// TwinCAT 3 PLC project PLC
// ProgramVersion: 3.1.4026.21
// libraries:
//   Core, * (Beckhoff Automation LLC)
//   CoreComponents, * (Beckhoff Automation LLC)
//   CoreMotionNc2, * (Beckhoff Automation LLC)
//   Tc2_ControllerToolbox, * (Beckhoff Automation GmbH)
//   Tc2_EtherCAT, * (Beckhoff Automation GmbH)
//   Tc2_MC2, * (Beckhoff Automation GmbH)
//   Tc2_Standard, * (Beckhoff Automation GmbH)
//   Tc2_System, * (Beckhoff Automation GmbH)
//   Tc2_TcpIp, * (Beckhoff Automation GmbH)
//   Tc3_JsonXml, * (Beckhoff Automation GmbH)
//   Tc3_PackML_V3, * (Beckhoff Automation GmbH)
// project tree:
//   AMR/ AMR_CONSTANT.TcGVL, AmrModule.TcPOU, AmrModule_HMI.TcPOU
//   AMR/DUT/ ST_AxisRecipe.TcDUT, ST_Recipe.TcDUT, ST_AmrModule_HMI.TcDUT
//   AMR/Interface/ I_AmrModule.TcIO
//   Components/Accelerometer %28EP3751%29/DUT/ ST_EP3751.TcDUT (not stored), ST_EP3751_HMI.TcDUT (not stored)
//   Components/Accelerometer %28EP3751%29/ EP3751_Accelerometer_HMI.TcPOU (not stored)
//   Components/ DEGREE_TO_RADIAN.TcPOU
//   Components/Encoder/DUT/ ST_EncoderConfig_HMI.TcDUT, ST_Encoder_HMI.TcDUT
//   Components/Encoder/ Encoder_HMI.TcPOU
//   Components/Nanotec/ COEDriveControl.TcPOU
//   Components/Nanotec/DUT/ ST_Nanotec_HMI.TcDUT
//   Components/Navitrol/Common types/ ST_SectionHeader.TcDUT, ST_SupervisorHeader.TcDUT
//   Components/Navitrol/HMI/ Navitrol_HMI.TcPOU, ST_Navitrol_HMI.TcDUT
//   Components/Navitrol/Interface/ I_Navitrol_DifferentialDriveMotorControl.TcIO, I_Navitrol_GoToDestination.TcIO, I_Navitrol_InitializePosition.TcIO, I_Navitrol_OmniDriveMotorControl.TcIO, I_Navitrol_ReturnToRoute.TcIO, I_Navitrol_Status.TcIO, I_Navitrol_StreamVelocity.TcIO
//   Components/Navitrol/ Msg1001_InitializePosition.TcPOU, Msg1016_MeasurmentUpdateDifferentialDrive.TcPOU, Msg3001_HoldRelease.TcPOU, Msg3002_NavitrolStatus.TcPOU, Msg3005_GoToDestination.TcPOU, Msg3024_ReturnToRoute.TcPOU, Navitrol_StreamVelocity.TcPOU
//   Components/Navitrol/Navitrol to Supervisor response/1100/ ST_1100_Position_initialization_started.TcDUT
//   Components/Navitrol/Navitrol to Supervisor response/1101/Components/ E_1101_Initialization_result.TcDUT
//   Components/Navitrol/Navitrol to Supervisor response/1101/ ST_1101_Position_initialized.TcDUT
//   Components/Navitrol/Navitrol to Supervisor response/1116/ ST_1116_Motor_Control_Differential.TcDUT
//   Components/Navitrol/Navitrol to Supervisor response/1126/Components/ ST_1126_Omni_wheels_ref_struct.TcDUT, ST_1126_Supervisor_status_out.TcDUT
//   Components/Navitrol/Navitrol to Supervisor response/1126/ ST_1126_Motor_control_omni_response.TcDUT
//   Components/Navitrol/Navitrol to Supervisor response/3101/ ST_3101_HoldReleased.TcDUT
//   Components/Navitrol/Navitrol to Supervisor response/3102/Components/ E_3102_Error_status.TcDUT, E_3102_Position_initialize_status.TcDUT, E_3102_State.TcDUT
//   Components/Navitrol/Navitrol to Supervisor response/3102/Components/Sections/1/ ST_3102_1_General_section.TcDUT
//   Components/Navitrol/Navitrol to Supervisor response/3102/ ST_3102_Navitrol_status.TcDUT
//   Components/Navitrol/Navitrol to Supervisor response/3105/ ST_3105_GoToDestinationResult.TcDUT
//   Components/Navitrol/Navitrol to Supervisor response/3124/ ST_3124_ReturnToRouteResponse.TcDUT
//   Components/Navitrol/Navitrol to Supervisor response/ U_Recived_bytes_from_Navitrol.TcDUT
//   Components/Navitrol/Supervisor to Navitrol message/1001/ ST_1001_Initialize_position.TcDUT
//   Components/Navitrol/Supervisor to Navitrol message/1016/ E_DriveControl.TcDUT, ST_1016_Measurement_update_differential_drive.TcDUT
//   Components/Navitrol/Supervisor to Navitrol message/1026/Components/ E_1026_Set_drive_mode.TcDUT, ST_1026_Omni_wheels_struct.TcDUT, ST_1026_Supervisor_status_bits.TcDUT
//   Components/Navitrol/Supervisor to Navitrol message/1026/ ST_1026_Measurement_update_generic_omni_drive.TcDUT
//   Components/Navitrol/Supervisor to Navitrol message/3001/ ST_3001_ReleaseHoldState.TcDUT
//   Components/Navitrol/Supervisor to Navitrol message/3002/Components/ E_3002_Set_ESTOP.TcDUT, E_3002_Status.TcDUT
//   Components/Navitrol/Supervisor to Navitrol message/3002/Components/Sections/2/Components/ E_3002_2_Enable_manual_control.TcDUT, E_3002_2_Inactive_Active.TcDUT
//   Components/Navitrol/Supervisor to Navitrol message/3002/Components/Sections/2/ ST_3002_2_Manual_section.TcDUT
//   Components/Navitrol/Supervisor to Navitrol message/3002/Components/Sections/6/Components/ E_3002_6_Joystick1_control_mode.TcDUT, E_3002_6_Joystick2_control_mode.TcDUT, E_3002_6_Steer_type_selection.TcDUT
//   Components/Navitrol/Supervisor to Navitrol message/3002/Components/Sections/6/ ST_3002_6_Remote_control_section.TcDUT
//   Components/Navitrol/Supervisor to Navitrol message/3002/Components/Sections/8/Components/ ST_3002_8_Binary_data.TcDUT, ST_3002_8_Error_status.TcDUT
//   Components/Navitrol/Supervisor to Navitrol message/3002/Components/Sections/8/ ST_3002_8_Battery_section.TcDUT
//   Components/Navitrol/Supervisor to Navitrol message/3002/Components/Sections/ F_SetSectionHeaderInfo.TcPOU
//   Components/Navitrol/Supervisor to Navitrol message/3002/ ST_3002_Supervisor_Status.TcDUT
//   Components/Navitrol/Supervisor to Navitrol message/3005/ ST_3005_GoToDestination.TcDUT
//   Components/Navitrol/Supervisor to Navitrol message/3024/ ST_3024_ReturnToRoute.TcDUT
//   Components/Navitrol/Supervisor to Navitrol message/ F_SetHeaderInfo.TcPOU
//   / MAIN.TcPOU, PlcTask.TcTTO
// real-time tasks:
//   TASK PlcTask: cycle T#2ms, priority 4, ADS port 350
// motion (NC):
//   TASK NC-Task 1 SAF: cycle T#4ms, priority 6, ADS port 501
//   TASK NC-Task 1 SVB: cycle T#4ms, priority 8, ADS port 511
//   AXIS WheelLeft (id 2)
//     General: UnitName=°
//     Dynamic: Acceleration=2708.277, Deceleration=2708.277, Jerk=8124.831
//     Velo: RefSearch=18.05518, RefSync=18.05518, SlowManual=90.2759, FastManual=541.6554, Fast=1805.518, Maximum=1805.518
//     OtherSettings: AllowMotionCmdToSlave=true
//     encoder EncType=19
//       EncPara: ScaleFactorNumerator=360, ScaleFactorDenominator=16777216, Inverse=true, MaxCount=#xffffffff
//     drive DrvType=16
//       DrvPara: Inverse=true, MaxCount=#xffffffff, DriveControlDWord=#x00020100
//         Analog: VeloReferenz=1986.0698, VeloScale=32, TorqueSetpointScale=10, ScaleFactorActTorque=0.1
//         TimeComp: TaskDelayCycles=1
//     controller CtrType=1
//       CtrPara: PriorControlFactor=1
//         Observer: BandWidth=20
//   AXIS WheelRight (id 3)
//     General: UnitName=°
//     Dynamic: Acceleration=2708.277, Deceleration=2708.277, Jerk=8124.831
//     Velo: RefSearch=18.05518, RefSync=18.05518, SlowManual=90.2759, FastManual=541.6554, Fast=1805.518, Maximum=1805.518
//     OtherSettings: AllowMotionCmdToSlave=true
//     encoder EncType=19
//       EncPara: ScaleFactorNumerator=360, ScaleFactorDenominator=16777216, MaxCount=#xffffffff
//     drive DrvType=16
//       DrvPara: MaxCount=#xffffffff, DriveControlDWord=#x00000100
//         Analog: VeloReferenz=1986.0698, VeloScale=32, TorqueSetpointScale=10, ScaleFactorActTorque=0.1
//         TimeComp: TaskDelayCycles=1
//     controller CtrType=1
//       CtrPara: PriorControlFactor=1
//         Observer: BandWidth=20
// I/O:
//   DEVICE X103 (EtherCAT), AmsNetId 0.0.0.0.3.1
//     EtherCat  (EK1100) [EK1100 EtherCAT Coupler (2A E-Bus)]
//       Motion 1 (ELM7231-9018) [ELM7231-9018 1Ch. Servo Terminal (48 V, 16 A RMS, OCT, STO, Safe Motion, TwinSAFE Logic)]
//         modules: Module 1 (SAFETY)
//       Motion 2 (ELM7231-9018) [ELM7231-9018 1Ch. Servo Terminal (48 V, 16 A RMS, OCT, STO, Safe Motion, TwinSAFE Logic)]
//         modules: Module 1 (SAFETY)
//       IO Link (EL6224-0090) [EL6224-0090 (IO Link Master, TwinSAFE SC)]
//         modules: Module 1 (DeviceState Inputs Device), Module 2 (DeviceState Inputs), Port1 (AHK5_14//ZIOB//16//BFR//), Module 4 (empty), Module 5 (empty), Module 6 (empty)
//       Safety PLC (EL2911) [EL2911, Potential supply terminal (10 A) with 4 Ch. Safety Inputs, TwinSAFE]
//         modules: Module 2 (FSOUT), Module 3 (DEVICEIO), Module 4 (FSLOGIC)
//       CAN Open (EL6751) [EL6751 CANopen Master]
//       Term 17 (EL9011) [EL9011 End Terminal]
//     Gyroscope (EP3751-0260) [EP3751-0260 Acceleration Sensor and Gyroscope]
//     Hokuyo Scanner (UAM-05LECA) [UAM-05LECA]
//       modules: Module 1 (Area Input Mode)
//   DEVICE CANOpen (EL6751), AmsNetId 0.0.0.0.6.1
//     Box 2 (PD4-CB59M024035-E-08)
// variable links:
//   (this object) <-> X103 (EtherCAT)/EtherCat  (EK1100)/Motion 1 (ELM7231-9018)
//     Drive/Inputs/In/nDataIn1 <-> DRV Following error actual value/Following error actual value
//     Drive/Inputs/In/nDcOutputTime <-> InfoData/DcOutputShift
//     Drive/Inputs/In/nState1 <-> DRV Statusword/Statusword
//     Drive/Inputs/In/nState2 <-> DRV Statusword/Statusword @bit 8
//     Drive/Inputs/In/nState4 @bit 1 <-> WcState/InputToggle0
//     Drive/Inputs/In/nState4 <-> WcState/WcState0
//     Drive/Outputs/Out/nCtrl1 <-> DRV Controlword/Controlword
//     Drive/Outputs/Out/nCtrl2 <-> DRV Controlword/Controlword @bit 8
//     Drive/Outputs/Out/nDataOut1 <-> DRV Target position/Target position
//     Enc/Inputs/In/nDataIn1 <-> FB Position/Position
//     Enc/Inputs/In/nDcInputTime <-> InfoData/DcInputShift
//     Enc/Inputs/In/nState4 @bit 1 <-> WcState/InputToggle0
//     Enc/Inputs/In/nState4 <-> WcState/WcState0
//     PlcTask Outputs/MAIN.AmrModule.SafetyResetELM.Reset <-> Module 1 (SAFETY)/SAFETY Standard Outputdata/FSOE/Connection ErrAck
//   (this object) <-> X103 (EtherCAT)/EtherCat  (EK1100)/Motion 2 (ELM7231-9018)
//     Drive/Inputs/In/nDataIn1 <-> DRV Following error actual value/Following error actual value
//     Drive/Inputs/In/nDcOutputTime <-> InfoData/DcOutputShift
//     Drive/Inputs/In/nState1 <-> DRV Statusword/Statusword
//     Drive/Inputs/In/nState2 <-> DRV Statusword/Statusword @bit 8
//     Drive/Inputs/In/nState4 @bit 1 <-> WcState/InputToggle0
//     Drive/Inputs/In/nState4 <-> WcState/WcState0
//     Drive/Outputs/Out/nCtrl1 <-> DRV Controlword/Controlword
//     Drive/Outputs/Out/nCtrl2 <-> DRV Controlword/Controlword @bit 8
//     Drive/Outputs/Out/nDataOut1 <-> DRV Target position/Target position
//     Enc/Inputs/In/nDataIn1 <-> FB Position/Position
//     Enc/Inputs/In/nDcInputTime <-> InfoData/DcInputShift
//     Enc/Inputs/In/nState4 @bit 1 <-> WcState/InputToggle0
//     Enc/Inputs/In/nState4 <-> WcState/WcState0
//     PlcTask Outputs/MAIN.AmrModule.SafetyResetELM.Reset <-> Module 1 (SAFETY)/SAFETY Standard Outputdata/FSOE/Connection ErrAck
//   (this object) <-> X103 (EtherCAT)
//     EtherCat  (EK1100)/Motion 2 (ELM7231-9018)/Module 1 (SAFETY)/SAFETY FSoE Connection 1 Receive Message/FSOE <-> EtherCat  (EK1100)/Safety PLC (EL2911)/ConnectionInputs/Motion.Motion 2 (ELM7231-9018) - Module 1 (SAFETY)_15 TxPDO
//     EtherCat  (EK1100)/Motion 2 (ELM7231-9018)/Module 1 (SAFETY)/SAFETY FSoE Connection 1 Send Message/FSOE <-> EtherCat  (EK1100)/Safety PLC (EL2911)/ConnectionOutputs/Motion.Motion 2 (ELM7231-9018) - Module 1 (SAFETY)_15 RxPDO
//     EtherCat  (EK1100)/Safety PLC (EL2911)/ConnectionInputs/Inputs.Hokuyo Scanner (UAM-05LECA) - Module 1 (Area Input Mode)_27 TxPDO <-> Hokuyo Scanner (UAM-05LECA)/Module 1 (Area Input Mode)/FSoE RxPDO-Map For Area Input Mode/FSOE
//     EtherCat  (EK1100)/Safety PLC (EL2911)/ConnectionInputs/Motion.Motion 2 (ELM7231-9018) - Module 1 (SAFETY)_15 TxPDO <-> EtherCat  (EK1100)/Motion 2 (ELM7231-9018)/Module 1 (SAFETY)/SAFETY FSoE Connection 1 Receive Message/FSOE
//     EtherCat  (EK1100)/Safety PLC (EL2911)/ConnectionOutputs/Inputs.Hokuyo Scanner (UAM-05LECA) - Module 1 (Area Input Mode)_27 RxPDO <-> Hokuyo Scanner (UAM-05LECA)/Module 1 (Area Input Mode)/FSoE TxPDO-Map For Area Input Mode/FSOE
//     EtherCat  (EK1100)/Safety PLC (EL2911)/ConnectionOutputs/Motion.Motion 2 (ELM7231-9018) - Module 1 (SAFETY)_15 RxPDO <-> EtherCat  (EK1100)/Motion 2 (ELM7231-9018)/Module 1 (SAFETY)/SAFETY FSoE Connection 1 Send Message/FSOE
//     Hokuyo Scanner (UAM-05LECA)/Module 1 (Area Input Mode)/FSoE RxPDO-Map For Area Input Mode/FSOE <-> EtherCat  (EK1100)/Safety PLC (EL2911)/ConnectionInputs/Inputs.Hokuyo Scanner (UAM-05LECA) - Module 1 (Area Input Mode)_27 TxPDO
//     Hokuyo Scanner (UAM-05LECA)/Module 1 (Area Input Mode)/FSoE TxPDO-Map For Area Input Mode/FSOE <-> EtherCat  (EK1100)/Safety PLC (EL2911)/ConnectionOutputs/Inputs.Hokuyo Scanner (UAM-05LECA) - Module 1 (Area Input Mode)_27 RxPDO
//   (this object) <-> CANOpen (EL6751)/Box 2 (PD4-CB59M024035-E-08)
//     PlcTask Inputs/MAIN.AmrModule.COEDriveControl.ActVel <-> TxPDO 3/Inputs/VarIn-0
//     PlcTask Inputs/MAIN.AmrModule.COEDriveControl.COEStatus <-> TxPDO 1/Inputs/VarIn-0
//     PlcTask Inputs/MAIN.AmrModule.COEDriveControl.ModeOfOperationStatus <-> TxPDO 1/Inputs/VarIn-1
//     PlcTask Outputs/MAIN.AmrModule.COEDriveControl.COEControl <-> RxPDO 1/Outputs/VarOut-0
//     PlcTask Outputs/MAIN.AmrModule.COEDriveControl.ModeOfOperation <-> RxPDO 1/Outputs/VarOut-1
//     PlcTask Outputs/MAIN.AmrModule.COEDriveControl.MotorTypeClosedLoop <-> RxPDO 1/Outputs/VarOut-2
//     PlcTask Outputs/MAIN.AmrModule.COEDriveControl.SetVel <-> RxPDO 3/Outputs/VarOut-0
//   (this object) <-> X103 (EtherCAT)/EtherCat  (EK1100)/IO Link (EL6224-0090)
//     PlcTask Inputs/MAIN.AmrModule.EncoderPositionIn <-> Port1 (AHK5_14//ZIOB//16//BFR//)/IO-Link Port1/Position
//     PlcTask Inputs/MAIN.AmrModule.EncoderSpeedIn <-> Port1 (AHK5_14//ZIOB//16//BFR//)/IO-Link Port1/Speed
//   (this object) <-> X103 (EtherCAT)/EtherCat  (EK1100)/Safety PLC (EL2911)
//     PlcTask Inputs/MAIN.AmrModule.SafetyEstop.InfoData/Diag <-> Function Block Info Data/Inputs.EStop.EStop1 Info Data/Diag
//     PlcTask Inputs/MAIN.AmrModule.SafetyEstop.InfoData/State <-> Function Block Info Data/Inputs.EStop.EStop1 Info Data/State
//     PlcTask Inputs/MAIN.AmrModule.SafetyInputGroup.InfoData/Diag <-> TwinSAFE Group Info Data/Inputs Info Data/Diag
//     PlcTask Inputs/MAIN.AmrModule.SafetyInputGroup.InfoData/State <-> TwinSAFE Group Info Data/Inputs Info Data/State
//     PlcTask Inputs/MAIN.AmrModule.SafetyMotionGroup.InfoData/Diag <-> TwinSAFE Group Info Data/Motion Info Data/Diag
//     PlcTask Inputs/MAIN.AmrModule.SafetyMotionGroup.InfoData/State <-> TwinSAFE Group Info Data/Motion Info Data/State
//     PlcTask Inputs/MAIN.AmrModule.SafetyScannerHokuyo.InfoData/Diag <-> Function Block Info Data/Inputs.AreaScanner.ScannerHokuyo Info Data/Diag
//     PlcTask Inputs/MAIN.AmrModule.SafetyScannerHokuyo.InfoData/State <-> Function Block Info Data/Inputs.AreaScanner.ScannerHokuyo Info Data/State
//     PlcTask Inputs/MAIN.AmrModule.SafetyScannerLeuze.InfoData/Diag <-> Function Block Info Data/Inputs.AreaScanner.ScannerLeuze Info Data/Diag
//     PlcTask Inputs/MAIN.AmrModule.SafetyScannerLeuze.InfoData/State <-> Function Block Info Data/Inputs.AreaScanner.ScannerLeuze Info Data/State
//     PlcTask Outputs/MAIN.AmrModule.SafetyGroupReset.Reset <-> StandardOutputs/Inputs.ErrorAcknowledgement_1
//     PlcTask Outputs/MAIN.AmrModule.SafetyGroupReset.Reset <-> StandardOutputs/Motion.ErrorAcknowledgement_13
//     PlcTask Outputs/MAIN.AmrModule.SafetyInputGroup.Run <-> StandardOutputs/Inputs.Run_18
//     PlcTask Outputs/MAIN.AmrModule.SafetyMotionGroup.Run <-> StandardOutputs/Motion.Run_20
//     PlcTask Outputs/MAIN.AmrModule.SafetyReset.Reset <-> StandardOutputs/Inputs.Reset_11
//     PlcTask Outputs/MAIN.AmrModule._BypassScanners <-> StandardOutputs/Inputs.BypassScanners_25
//   (this object) <-> X103 (EtherCAT)/Gyroscope (EP3751-0260)
//     PlcTask Inputs/MAIN.AmrModule.EP3751_IO/ACC_X <-> AI Acc X Samples 1 (Real32)/Samples[0]
//     PlcTask Inputs/MAIN.AmrModule.EP3751_IO/ACC_Y <-> AI Acc Y Samples 1 (Real32)/Samples[0]
//     PlcTask Inputs/MAIN.AmrModule.EP3751_IO/ACC_Z <-> AI Acc Z Samples 1 (Real32)/Samples[0]
//     PlcTask Inputs/MAIN.AmrModule.EP3751_IO/Gyro_X <-> AI Gyro X Samples 1 (Real32)/Samples[0]
//     PlcTask Inputs/MAIN.AmrModule.EP3751_IO/Gyro_Y <-> AI Gyro Y Samples 1 (Real32)/Samples[0]
//     PlcTask Inputs/MAIN.AmrModule.EP3751_IO/Gyro_Z <-> AI Gyro Z Samples 1 (Real32)/Samples[0]
//   (this object) <-> NC-Task 1 SAF/Axes/WheelLeft
//     PlcTask Inputs/MAIN.AmrModule.WheelLeftRef.NcToPlc <-> Outputs/ToPlc
//     PlcTask Outputs/MAIN.AmrModule.WheelLeftRef.PlcToNc <-> Inputs/FromPlc
//   (this object) <-> NC-Task 1 SAF/Axes/WheelRight
//     PlcTask Inputs/MAIN.AmrModule.WheelRightRef.NcToPlc <-> Outputs/ToPlc
//     PlcTask Outputs/MAIN.AmrModule.WheelRightRef.PlcToNc <-> Inputs/FromPlc

CONFIGURATION PLC
    RESOURCE PLC ON TwinCAT3
        TASK PlcTask(INTERVAL := T#2ms, PRIORITY := 4);
        PROGRAM MAIN WITH PlcTask : MAIN;
    END_RESOURCE
END_CONFIGURATION

// ---- AMR/DUT/ST_AxisRecipe.TcDUT
TYPE ST_AxisRecipe :
	STRUCT
		Velocity	 : LREAL := 10;
		Acceleration : LREAL := 1000;
		Deceleration : LREAL := 1000;
		Jerk		 : LREAL := 1000;
	END_STRUCT
END_TYPE

// ---- AMR/DUT/ST_Recipe.TcDUT
TYPE ST_Recipe :
	STRUCT
		LiftPosition_Up	  : LREAL := 100;
		LiftPosition_Down : LREAL := 0;
	END_STRUCT
END_TYPE

// ---- AMR/DUT/ST_AmrModule_HMI.TcDUT
TYPE ST_AmrModule_HMI :
	STRUCT
		Override	   : LREAL := 100.0;
		BypassScanners : BOOL  := TRUE;
	END_STRUCT
END_TYPE

// ---- Components/Encoder/DUT/ST_EncoderConfig_HMI.TcDUT
TYPE ST_EncoderConfig_HMI :
	STRUCT
		Speed_InputMinimum	   : LREAL := -32768;
		Speed_InputMaximum	   : LREAL := 32767;
		Speed_OutputMinimum	   : LREAL := -32768;
		Speed_OutputMaximum	   : LREAL := 32767;
		Position_InputMinimum  : LREAL := -32768;
		Position_InputMaximum  : LREAL := 32767;
		Position_OutputMinimum : LREAL := -32768;
		Position_OutputMaximum : LREAL := 32767;
	END_STRUCT
END_TYPE

// ---- Components/Encoder/DUT/ST_Encoder_HMI.TcDUT
TYPE ST_Encoder_HMI EXTENDS ST_HmiFunction :
	STRUCT
		Config			 : ST_EncoderConfig_HMI;
		ActualSpeed		 : LREAL;
		ActualPosition	 : LREAL;
		RawValueSpeed	 : INT;
		RawValuePosition : UINT;
	END_STRUCT
END_TYPE

// ---- Components/Nanotec/DUT/ST_Nanotec_HMI.TcDUT
TYPE ST_Nanotec_HMI EXTENDS ST_HmiFunction :
	STRUCT
		JogFwd	   : Button;
		JogBwd	   : Button;
		Ready	   : BOOL;
		Faulted	   : BOOL;
		ActVelIncr : INT;
	END_STRUCT
END_TYPE

// ---- Components/Navitrol/Common types/ST_SectionHeader.TcDUT
{attribute 'pack_mode' := '1'}
TYPE ST_SectionHeader :
	STRUCT
		Section_ID	   : UINT;
		Section_length : UDINT;
	END_STRUCT
END_TYPE

// ---- Components/Navitrol/Common types/ST_SupervisorHeader.TcDUT
{attribute 'pack_mode' := '1'}

//{attribute 'hide_all_locals'}
TYPE ST_SupervisorHeader :
	STRUCT
		Protocol_version : UINT;
		Message_ID		 : UINT;
		Message_length	 : UDINT;
	END_STRUCT
END_TYPE

//When sending a message from Supervisor to Navitrol, this is populated using F_SetHeaderInfo.

// ---- Components/Navitrol/HMI/ST_Navitrol_HMI.TcDUT
TYPE ST_Navitrol_HMI EXTENDS ST_HmiFunction :
	STRUCT
		CommunicationActive : BOOL;
		Status				: E_3102_State;
		ControlFromNavitrol : BOOL;
	END_STRUCT
END_TYPE

// ---- Components/Navitrol/Navitrol to Supervisor response/1100/ST_1100_Position_initialization_started.TcDUT
{attribute 'pack_mode' := '1'}
TYPE ST_1100_Position_initialization_started EXTENDS ST_SupervisorHeader :
	STRUCT
	END_STRUCT
END_TYPE

// ---- Components/Navitrol/Navitrol to Supervisor response/1101/Components/E_1101_Initialization_result.TcDUT
{attribute 'qualified_only'}
{attribute 'strict'}
{attribute 'to_string'}
TYPE E_1101_Initialization_result : (
		Failure := 0,
		Success := 1
	) UINT;
END_TYPE

//0 - Failure

//	The position initialization can fail for example if

//		- A good position is not found within pos_ini_max_d..-parameters from the given pos init point

//		- A good position is not found within value of pos_init_max_wait_time-parameter

//		- The AGV is not stationary state, it is performing load or there are scanner related errors active.

//1 - Success

//		- A good position was found near the given position initialization point and position was successfully initialized.

// ---- Components/Navitrol/Navitrol to Supervisor response/1101/ST_1101_Position_initialized.TcDUT
{attribute 'pack_mode' := '1'}
TYPE ST_1101_Position_initialized EXTENDS ST_SupervisorHeader :
	STRUCT
		X					  : REAL;  //	X-map coordinate OF the new position in meters
		Y					  : REAL;  //	Y-map coordinate of the new position in meters
		H					  : REAL;  //	Heading of the new position on the map in radians
		Floor				  : UDINT; //		The floor of the new position
		Initialization_result : E_1101_Initialization_result;
		Position_confidence	  : UINT; //		Position confidence percentage (1 - 100%)Describes how well the laser measurements in the new position matches the seen environment.	
	END_STRUCT
END_TYPE

// ---- Components/Navitrol/Navitrol to Supervisor response/1116/ST_1116_Motor_Control_Differential.TcDUT
{attribute 'pack_mode' := '1'}
TYPE ST_1116_Motor_Control_Differential EXTENDS ST_SupervisorHeader :
	STRUCT
		Message_number			: UDINT; //Identification number for individual messages. NOTE: This value must match with the latest Odometer update message number sent by the Supervisor.
		Speed_Left				: REAL;	 // Reference speed for left wheel (m/s)
		Speed_Right				: REAL;	 // Reference speed for right wheel (m/s)
		Errors_Stopping_driving : UINT;	 //0 no errors, 1 error stopping driving
	END_STRUCT
END_TYPE

// ---- Components/Navitrol/Navitrol to Supervisor response/1126/Components/ST_1126_Omni_wheels_ref_struct.TcDUT
{attribute 'pack_mode' := '1'}
TYPE ST_1126_Omni_wheels_ref_struct :
	STRUCT
		Steer_angle_reference : REAL;
		Wheel_speed_reference : REAL;
	END_STRUCT
END_TYPE

// ---- Components/Navitrol/Navitrol to Supervisor response/1126/Components/ST_1126_Supervisor_status_out.TcDUT
{attribute 'pack_mode' := '1'}
TYPE ST_1126_Supervisor_status_out :
	STRUCT
		Navitrol_error : BIT; //	Navitrol has ANY error active AND is unable TO drive.
		Reserved_1	   : BIT;
		Reserved_2	   : BIT;
		Reserved_3	   : BIT;
		Reserved_4	   : BIT;
		Reserved_5	   : BIT;
		Reserved_6	   : BIT;
		Brake_release  : BIT;  //	Navitrol requests Supevisor to release brakes to start driving
		Reserved	   : BYTE; //	Not in use	
	END_STRUCT
END_TYPE

// ---- Components/Navitrol/Navitrol to Supervisor response/1126/ST_1126_Motor_control_omni_response.TcDUT
{attribute 'pack_mode' := '1'}
TYPE ST_1126_Motor_control_omni_response EXTENDS ST_SupervisorHeader :
	STRUCT
		Message_number		   : UDINT;
		Supervisor_status_out  : ST_1126_Supervisor_status_out;
		Driving_vector_Angle   : REAL; //Reference driving vector angle relative to the vehicle frame. (+/-PI in radians)0-forwards along vehicle center line. Positive direction is CCW from vehicle center lin
		Steering_Radius		   : REAL; //Radius to center of rotation from navigation point (m).0-pivoting around vehicle navigation point. Positive value sets the center of rotation to a direction of 90 deg CCW from the driving vector angle. For example with 0 deg driving vector angle vehicle turns to left with positive radius and to right with negative radius.
		Navigation_point_speed : REAL; //Reference speed of the vehicle navigation point along driving vector (m/s) Positive along driving vector, negative against driving vector (i.e. driving vector ± PI).
		Number_of_Wheels	   : UINT; //Number of omni wheels, maximum 6, minimum 2. Determined by parameter omni_steer_nbr
		Omni_wheels_ref_struct : ARRAY[0..1] OF
			ST_1126_Omni_wheels_ref_struct; //The references for each individual omni wheel
	END_STRUCT
END_TYPE

// ---- Components/Navitrol/Navitrol to Supervisor response/3101/ST_3101_HoldReleased.TcDUT
TYPE ST_3101_HoldReleased EXTENDS ST_SupervisorHeader :
	STRUCT
		ReleaseStopHoldResult : UINT;
	END_STRUCT
END_TYPE

// ---- Components/Navitrol/Navitrol to Supervisor response/3102/Components/E_3102_Error_status.TcDUT
{attribute 'qualified_only'}
{attribute 'strict'}
{attribute 'to_string'}
TYPE E_3102_Error_status : (
		no_error := 0,
		error_on := 1
	) UINT;
END_TYPE

// ---- Components/Navitrol/Navitrol to Supervisor response/3102/Components/E_3102_Position_initialize_status.TcDUT
{attribute 'qualified_only'}
{attribute 'strict'}
{attribute 'to_string'}
TYPE E_3102_Position_initialize_status : (
		Failed	  := 0,
		Succeeded := 1
	) UINT;
END_TYPE

// ---- Components/Navitrol/Navitrol to Supervisor response/3102/Components/E_3102_State.TcDUT
{attribute 'qualified_only'}
{attribute 'strict'}
{attribute 'to_string'}
TYPE E_3102_State : //Navitrol state
	(
		INVALID		  := 0,
		START_STATE	  := 1,
		STANDBY_STATE := 2,
		AUTO_STATE	  := 3,
		FSTOP_STATE	  := 9,
		LOAD_STATE	  := 14,
		HOLD_STATE	  := 15,
		MANUAL_STATE  := 16,
		PAUSE_STATE	  := 17
	) UDINT;
END_TYPE

// ---- Components/Navitrol/Navitrol to Supervisor response/3102/Components/Sections/1/ST_3102_1_General_section.TcDUT
{attribute 'pack_mode' := '1'}
TYPE ST_3102_1_General_section EXTENDS ST_SectionHeader :
	STRUCT
		Battery_voltage : REAL; // V
		On_route		: UINT; // 1 on route, 0 not on route
	END_STRUCT
END_TYPE

// ---- Components/Navitrol/Navitrol to Supervisor response/3102/ST_3102_Navitrol_status.TcDUT
{attribute 'pack_mode' := '1'}
TYPE ST_3102_Navitrol_status EXTENDS ST_SupervisorHeader :
	STRUCT
		DefaultSectionLength	   : UDINT;
		State					   : E_3102_State;
		X_coordinate			   : REAL; //In meters
		Y_coordinate			   : REAL; //In meters
		Heading					   : REAL; //Radians
		Level					   : DINT; //Level ID
		Speed					   : REAL; //m/s
		Position_initialize_status : E_3102_Position_initialize_status;
		Position_confidence		   : UINT; //Position confidence in percentage (1 - 100%)
		Error_status			   : E_3102_Error_status;
		//Additional sections can be added bellow - based on what is requested in the array of ST_3002_Supervisor_Status.Section_IDs 
		General_section : ST_3102_1_General_section;
	END_STRUCT
END_TYPE

// ---- Components/Navitrol/Navitrol to Supervisor response/3105/ST_3105_GoToDestinationResult.TcDUT
TYPE ST_3105_GoToDestinationResult EXTENDS ST_SupervisorHeader :
	STRUCT
		DestinationID : UDINT;
		GoToResult	  : UDINT;
	END_STRUCT
END_TYPE

// ---- Components/Navitrol/Navitrol to Supervisor response/3124/ST_3124_ReturnToRouteResponse.TcDUT
TYPE ST_3124_ReturnToRouteResponse EXTENDS ST_SupervisorHeader :
	STRUCT
        ReturnToRouteResult : UDINT;
	END_STRUCT
END_TYPE

// ---- Components/Navitrol/Navitrol to Supervisor response/U_Recived_bytes_from_Navitrol.TcDUT
// Bytes bucket to buffer received messages.

// Header info is parsed before being copied into the correct message structure.

// PLC logic is built expecting to receive the entire TCP message payload with one call to FB_SocketReceive.

// FB_SocketReceive will fragment the received data if the receive buffer is not large enough.

// Make sure this is large enough to fit the biggest received message.
TYPE U_Recived_bytes_from_Navitrol : UNION
		Header : ST_SupervisorHeader;
		Bytes  : ARRAY[0..2047] OF UINT;
	END_UNION
END_TYPE

// ---- Components/Navitrol/Supervisor to Navitrol message/1001/ST_1001_Initialize_position.TcDUT
{attribute 'pack_mode' := '1'}
TYPE ST_1001_Initialize_position EXTENDS ST_SupervisorHeader :
	STRUCT
		X	  : REAL; //		X - map coordinate OF the AGV in meters
		Y	  : REAL; //		Y - map coordinate of the AGV in meters
		H	  : REAL; //		Heading of the AGV on the map in radians
		Level : DINT; //	The level ID on which the AGV is located
	END_STRUCT
END_TYPE

// ---- Components/Navitrol/Supervisor to Navitrol message/1016/E_DriveControl.TcDUT
{attribute 'qualified_only'}
{attribute 'strict'}
{attribute 'to_string'}
TYPE E_DriveControl : (
		Idle := 0,
		Activate_auto_mode,
		Activate_supervisor_error,
		Activate_manual_mode,
		Activate_emergency_stop
	) UINT;
END_TYPE

// ---- Components/Navitrol/Supervisor to Navitrol message/1016/ST_1016_Measurement_update_differential_drive.TcDUT
{attribute 'pack_mode' := '1'}
TYPE ST_1016_Measurement_update_differential_drive EXTENDS ST_SupervisorHeader :
	STRUCT
		Message_number		 : UDINT;
		Odometry_left_wheel	 : UDINT; // The cumulative encoder value from the left wheel. The scale from encoder value to meters is defined by mot_ctrl_left_dist_scale-parameter The overflow point must be from 0xffffffff to 0
		Odometry_right_wheel : UDINT;
		Drive_control		 : E_DriveControl := E_DriveControl.Activate_auto_mode;
		Timestamp			 : UDINT; // Cumulative time in milliseconds. Time base can be chosen freely.
	END_STRUCT
END_TYPE

// ---- Components/Navitrol/Supervisor to Navitrol message/1026/Components/E_1026_Set_drive_mode.TcDUT
{attribute 'qualified_only'}
{attribute 'strict'}
{attribute 'to_string'}
TYPE E_1026_Set_drive_mode : (
		Manual_mode	   := 1,
		Automatic_mode := 2
	) UINT;
END_TYPE

// ---- Components/Navitrol/Supervisor to Navitrol message/1026/Components/ST_1026_Omni_wheels_struct.TcDUT
{attribute 'pack_mode' := '1'}
TYPE ST_1026_Omni_wheels_struct :
	STRUCT
		Steer_angle : REAL;
		Wheel_speed : REAL;
	END_STRUCT
END_TYPE

// ---- Components/Navitrol/Supervisor to Navitrol message/1026/Components/ST_1026_Supervisor_status_bits.TcDUT
{attribute 'pack_mode' := '1'}
TYPE ST_1026_Supervisor_status_bits :
	STRUCT
		Error		   : BIT;  //	When active ERROR_MOTOR_CONTROL_FAULT will be set.See error. in Glossary
		Emergency_stop : BIT;  //	When active Navitrol will perform emergency stop and following two warnings will be triggered: WARNING_AGV_EM_STOP and WARNING_ESTOP_ACTIVE
		Soft_slow	   : BIT;  //	When active Navitrol will perform soft slow.
		Soft_stop	   : BIT;  //	When active Navitrol will perform soft stop.
		Reserved_4	   : BIT;  //Not in use
		Reserved_5	   : BIT;  //Not in use
		Reserved_6	   : BIT;  //Not in use
		Brake_released : BIT;  //	Informs Navitrol of the status of brakes.When not active hard stop will be enabled.
		Reserved_8_15  : BYTE; // Not in use
	END_STRUCT
END_TYPE

// ---- Components/Navitrol/Supervisor to Navitrol message/1026/ST_1026_Measurement_update_generic_omni_drive.TcDUT
{attribute 'pack_mode' := '1'}
TYPE ST_1026_Measurement_update_generic_omni_drive EXTENDS ST_SupervisorHeader :
	STRUCT
		Message_number	  : UDINT;
		Set_drive_mode	  : E_1026_Set_drive_mode;
		Supervisor_status : ST_1026_Supervisor_status_bits			  := (Brake_released := TRUE);
		Number_of_wheels  : UINT									  := 2;
		Omni_wheels		  : ARRAY[0..1] OF ST_1026_Omni_wheels_struct := [2((Steer_angle := 0.1))];
	END_STRUCT
END_TYPE

// ---- Components/Navitrol/Supervisor to Navitrol message/3001/ST_3001_ReleaseHoldState.TcDUT
TYPE ST_3001_ReleaseHoldState EXTENDS ST_SupervisorHeader :
	STRUCT
		DestinationId : UDINT := 0;
	END_STRUCT
END_TYPE

// ---- Components/Navitrol/Supervisor to Navitrol message/3002/Components/E_3002_Set_ESTOP.TcDUT
{attribute 'qualified_only'}
{attribute 'strict'}
{attribute 'to_string'}
TYPE E_3002_Set_ESTOP : (
		Release_ESTOP := 0,
		Set_ESTOP	  := 1
	) UINT;
END_TYPE

// ---- Components/Navitrol/Supervisor to Navitrol message/3002/Components/E_3002_Status.TcDUT
{attribute 'qualified_only'}
{attribute 'strict'}
{attribute 'to_string'}
TYPE E_3002_Status : (
		Not_ok := 0, //ERROR_PLC_FAILURE will be activated, and additionally manual driving will be prevented.
		Ok	   := 1	 //Navitrol is allowed to drive the AGV.
	) UINT;
END_TYPE

// ---- Components/Navitrol/Supervisor to Navitrol message/3002/Components/Sections/2/Components/E_3002_2_Enable_manual_control.TcDUT
{attribute 'qualified_only'}
{attribute 'strict'}
{attribute 'to_string'}
TYPE E_3002_2_Enable_manual_control : (
		Enable_control	:= 0,
		Disable_control := 1
	) UINT;
END_TYPE

(*
Used to enable manual control from this section:
	0 - Enable control
Navitrol will activate manual mode and sets WARNING_ETH_MANUAL_MODE. This section can be used to drive the AGV.
	1 - Disable control
Navitrol will ignore any controls from this section.
*)

// ---- Components/Navitrol/Supervisor to Navitrol message/3002/Components/Sections/2/Components/E_3002_2_Inactive_Active.TcDUT
{attribute 'qualified_only'}
{attribute 'strict'}
{attribute 'to_string'}
TYPE E_3002_2_Inactive_Active : (
		Inactive := 0,
		Active	 := 1
	) UINT;
END_TYPE

// ---- Components/Navitrol/Supervisor to Navitrol message/3002/Components/Sections/2/ST_3002_2_Manual_section.TcDUT
{attribute 'pack_mode' := '1'}
TYPE ST_3002_2_Manual_section EXTENDS ST_SectionHeader :
	STRUCT
		Enable_manual_control : E_3002_2_Enable_manual_control;
		Forward				  : E_3002_2_Inactive_Active;
		Backward			  : E_3002_2_Inactive_Active;
		Left				  : E_3002_2_Inactive_Active;
		Right				  : E_3002_2_Inactive_Active;
		Drive_speed			  : REAL; //The manual drive speed reference in meters per second.
	END_STRUCT
END_TYPE

// ---- Components/Navitrol/Supervisor to Navitrol message/3002/Components/Sections/6/Components/E_3002_6_Joystick1_control_mode.TcDUT
{attribute 'qualified_only'}
{attribute 'strict'}
{attribute 'to_string'}
TYPE E_3002_6_Joystick1_control_mode : (
		No_control	   := 0,
		Old_control	   := 1,
		Vector_control := 2
	) UINT;
END_TYPE

(*
Selects the joystick 1 control mode:
	0 - No control
Joystick 1 x and y values are ignored.
	1 - Old control
	Not recommended
	Navitrol activates manual mode. Curvature is calculated directly from joystick 1 x value and the speed from joystick 1 y value.
2 - Vector control
	Recommended
	Navitrol activates manual mode. A unit vector is calculated from joystick 1 xy-values. The speed comes from the length of the vector (Positive when y is positive) and the curvature from its angle from the Y-axis.
	For example AGV drives forward and curves right when x and y are positive.
	For more information, see "Joystick System" chapter from Web Interface document

*)

// ---- Components/Navitrol/Supervisor to Navitrol message/3002/Components/Sections/6/Components/E_3002_6_Joystick2_control_mode.TcDUT
{attribute 'qualified_only'}
{attribute 'strict'}
{attribute 'to_string'}
TYPE E_3002_6_Joystick2_control_mode : (
		No_control			:= 0,
		Enable_lift_control := 1
	) UINT;
END_TYPE

(*
Selects the joystick 2 control mode:
	0 - No control
Joystick 1 x and y values are ignored.
	1 - Enable lift control
	Navitrol activates manual mode.
*)

// ---- Components/Navitrol/Supervisor to Navitrol message/3002/Components/Sections/6/Components/E_3002_6_Steer_type_selection.TcDUT
{attribute 'qualified_only'}
{attribute 'strict'}
{attribute 'to_string'}
TYPE E_3002_6_Steer_type_selection : (
		Invalid					:= 0,
		Front_wheel_steer		:= 1,
		Mid_wheel_steer			:= 2,
		Rear_wheel_steer		:= 3,
		Pivot_steer				:= 5,
		Parallel_steer_forward	:= 6,
		Parallel_steer_backward := 7
	);
END_TYPE

(*
1 - Front wheel steer
Only for omni drives. Moves the navigation point to between the front wheels. With this steer type almost all turning control will be done by the rear wheels.
2 - Mid wheel steer
	Normal driving. The normal navigation point is used.
3 - Rear wheel steer
	Only for omni drives. Moves the navigation point to between the rear wheels. With this steer type almost all turning control will be done by the front wheels.
5 - Pivot steer
	Pivot curvature is always given, and supervisor can control only the speed up to maximum of pivot_speed-parameter. This mode should only be activated, if the AGV can pivot.
6 - Parallel steer forward
	Only for omni drives.
	The curvature in this mode is always zero. Instead of curvature supervisor controls the frame heading instead and speed. Wheels will rotate forward with positive speed reference.
7 - Parallel steer backward
	Only for omni drives.
	The curvature in this mode is always zero. Instead of curvature supervisor controls the frame heading instead and speed. Wheels will rotate backwards with positive speed reference.

*)

// ---- Components/Navitrol/Supervisor to Navitrol message/3002/Components/Sections/6/ST_3002_6_Remote_control_section.TcDUT
{attribute 'pack_mode' := '1'}
TYPE ST_3002_6_Remote_control_section EXTENDS ST_SectionHeader :
	STRUCT
		Joystick1_control_mode : E_3002_6_Joystick1_control_mode;
		Joystick1_x			   : REAL;
		Joystick1_y			   : REAL;
		Joystick2_control_mode : E_3002_6_Joystick2_control_mode;
		Joystick2_x			   : REAL; //0 - Not in use
		Joystick2_y			   : REAL; (*Lift actuator height reference control.
										If the given y-value is larger than 0.1 actuator control is enabled. 
										And the y-value is scaled with actuator_eth_ctrl_scale-parameter and added to the previous actuator reference. 
										The actuator reference can be controlled only between values of actuator_min_val and actuator_max_val parameters.Valid values [-1...1]*)
		Steer_type_selection : E_3002_6_Steer_type_selection;
	END_STRUCT
END_TYPE

// ---- Components/Navitrol/Supervisor to Navitrol message/3002/Components/Sections/8/Components/ST_3002_8_Binary_data.TcDUT
{attribute 'pack_mode' := '1'}
TYPE ST_3002_8_Binary_data :
	STRUCT
		Request_charge	 : BIT; // This charge request info is show in motor control messages and in Navitrol battery status section if charging_cmd_source-parameter is set to 3. No drive orders or other actions are made based on this.
		Charging_active	 : BIT; // Informs Navitrol that charging is active. Navitrol will set soft stop (parameter charging_prevents_driving).
		Balancing_active : BIT; // Informs Navitrol that battery balancing is active at charger. Navitrol will set soft stop (parameter charging_prevents_driving).
		Reserved_3		 : BIT; // 0 - Not in use
		Reserved_4		 : BIT; // 0 - Not in use
		Reserved_5		 : BIT; // 0 - Not in use
		Reserved_6		 : BIT; // 0 - Not in use
		Reserved_7		 : BIT; // 0 - Not in use
	END_STRUCT
END_TYPE

// ---- Components/Navitrol/Supervisor to Navitrol message/3002/Components/Sections/8/Components/ST_3002_8_Error_status.TcDUT
{attribute 'pack_mode' := '1'}
TYPE ST_3002_8_Error_status :
	STRUCT
		Communication_error		  : BIT; // BMS has lost the communication to the battery. *
		Configuration_error		  : BIT; // Battery has not been correctly configured. *
		Undervoltage			  : BIT; // Undervoltage detected. Operating voltage is low. Prepare to charge or replace the battery. *
		Overvoltage				  : BIT; // Overvoltage detected. Overvoltage is a sustained voltage that exceeds the normal steady state limits. *
		Overcurrent				  : BIT; // Overcurrent detected. Might be caused by overloading or short circuiting the battery. *
		Temperature_error		  : BIT; // The temperature of the battery is at unsafe levels. * In addition, Navitrol will set ERROR_BATTERY_HIGH_TEMPERATURE
		Internal_defect			  : BIT; // The battery has a defect and might not work properly. *
		Bad_state_of_health		  : BIT; // The battery is worn down in use. It might not fully charge anymore. *
		Faulty_charger			  : BIT; // The charger connected to the battery is not working. *
		Faulty_contactor		  : BIT; // The contactor of the battery is not working. *
		Current_sensor_defect	  : BIT; // The current sensor of the battery is not working. *
		Temperature_sensor_defect : BIT; // The temperature sensor of the battery is not working. *
		Battery_cell_drift		  : BIT; // Two or more battery cells are in imbalance. Can lead to over-charging or over-discharging harming the battery. *
		Charging_error			  : BIT; // Error while charging the battery *
		Generic_error			  : BIT; // This can be used to indicate that there is some other battery related error that is not listed above. *
		Reserved				  : BIT; // 0 - Not in use
	END_STRUCT
END_TYPE

// ---- Components/Navitrol/Supervisor to Navitrol message/3002/Components/Sections/8/ST_3002_8_Battery_section.TcDUT
{attribute 'pack_mode' := '1'}
TYPE ST_3002_8_Battery_section EXTENDS ST_SectionHeader :
	STRUCT
		// Battery state of charge percentage. Valid values [0...100] 65535 - Not available

		// This will be used for determining the battery level if battery_percentage_from_mot_ctrl-parameter is set to 1.
		State_of_charge : UINT := 100;
		// Battery voltage in 0.1 Volts. For example, 4.2V would be 42 65535 - Not available

		// This will be used for determining the battery level if battery_percentage_from_mot_ctrl-parameter is set to 0.
		Voltage : UINT := 42;
		// Charge current / current draw in 0.1 Amperes. Negative values when battery is discharging

		// and positive values when battery is being charged. 32767 - Not available

		// Only for statistics - visible in Navitrol Monitor.
		Charge_current_draw : INT := 10;
		// Energy draw in 0.1 Ampere hours Negative values when battery is discharging

		// and positive values when battery is being charged. 32767 - Not available

		// Only for statistics - visible in Navitrol Monitor.
		Energy_draw : INT := 100;
		// Estimated time left in minutes until the battery is empty. 65535 - Not available

		// Only for statistics - visible in Navitrol Monitor.
		Time_remaining : UINT := 45;
		// Battery state of health percentage. Describes the overall state of the battery. Valid values [0...100] 65535 - Not available

		// Only for statistics - visible in Navitrol Monitor.
		State_of_health : UINT := 100;
		// Battery temperature in Celsius degrees. 32767 - Not available

		// Used to trigger WARNING_BATTERY_HIGH_TEMPERATURE if given temperature is larger than

		// battery_high_temperature_warning_limit_C and ERROR_BATTERY_HIGH_TEMPERATURE if larger

		// than battery_high_temperature_error_limit_C
		Temperature : INT := 32;
		// Total number of load cycles performed for the battery. 65535 - Not available

		// Only for statistics - visible in Navitrol Monitor.
		Load_cycle_count : UINT := 20;
		// Total number of operating hours of the battery. 65535 - Not available

		// Only for statistics - visible in Navitrol Monitor.
		Operating_hours : UINT := 155;
		// Voltage of the charger in 0.1 Volts. 65535 - Not available

		// Only for statistics - visible in Navitrol Monitor.
		Charger_voltage : UINT := 420;
		// Error status information. If any of the errors marked with * are active Navitrol Monitor will view its description

		// and Navitrol set WARNING_BATTERY_ERROR_OR_WARNING_ACTIVE 0 - No error
		Error_status : ST_3002_8_Error_status;
		// Battery related binary data and requests 0 - Inactive
		Binary_data : ST_3002_8_Binary_data;
		// 0 - Not in use
		Reserved : BYTE;
	END_STRUCT
END_TYPE

// ---- Components/Navitrol/Supervisor to Navitrol message/3002/ST_3002_Supervisor_Status.TcDUT
{attribute 'pack_mode' := '1'}
TYPE ST_3002_Supervisor_Status EXTENDS ST_SupervisorHeader :
	STRUCT
		Status			   : E_3002_Status			  := E_3002_Status.Ok;
		Set_Estop		   : E_3002_Set_ESTOP		  := E_3002_Set_ESTOP.Release_ESTOP;
		Number_of_sections : UINT					  := 1;	  //Number of sections requested in response message 3102. Change the size of Section_IDs's bellow to match.
		Section_IDs		   : ARRAY[1..1] OF UINT	  := [1]; //List of sections requested to send in the response message 3102. Make sure to add the expected recived message sections to the end of ST_3102_Navitrol_status
		Manual_section	   : ST_3002_2_Manual_section := (Enable_manual_control := E_3002_2_Enable_manual_control.Disable_control);
		Battery_section	   : ST_3002_8_Battery_section;
	END_STRUCT
END_TYPE

// ---- Components/Navitrol/Supervisor to Navitrol message/3005/ST_3005_GoToDestination.TcDUT
TYPE ST_3005_GoToDestination EXTENDS ST_SupervisorHeader :
	STRUCT
		DestinationID : UDINT;
	END_STRUCT
END_TYPE

// ---- Components/Navitrol/Supervisor to Navitrol message/3024/ST_3024_ReturnToRoute.TcDUT
TYPE ST_3024_ReturnToRoute EXTENDS ST_SupervisorHeader :
	STRUCT
	END_STRUCT
END_TYPE

// ---- AMR/AMR_CONSTANT.TcGVL
{attribute 'qualified_only'}
VAR_GLOBAL CONSTANT
	WHEEL_DIAMETER : LREAL := 0.160; // Wheel Diameter in m
END_VAR

// ---- AMR/Interface/I_AmrModule.TcIO
INTERFACE I_AmrModule EXTENDS I_Module, I_Override, I_ContainStatemachine

PROPERTY BypassScanners : BOOL
SET
END_SET
END_PROPERTY

METHOD ResetSafety
END_METHOD

PROPERTY WheelLeft : I_Axis_PTP
GET
END_GET
END_PROPERTY

PROPERTY WheelLeftStreamVelocity : I_Navitrol_StreamVelocity
GET
END_GET
END_PROPERTY

PROPERTY WheelRight : I_Axis_PTP
GET
END_GET
END_PROPERTY

PROPERTY WheelRightStreamVelocity : I_Navitrol_StreamVelocity
GET
END_GET
END_PROPERTY

END_INTERFACE

// ---- Components/Navitrol/Interface/I_Navitrol_DifferentialDriveMotorControl.TcIO
INTERFACE I_Navitrol_DifferentialDriveMotorControl EXTENDS I_Base

{attribute 'monitoring' := 'call'}
PROPERTY EncoderCountWheelLeft : UDINT
SET
END_SET
END_PROPERTY

{attribute 'monitoring' := 'call'}
PROPERTY EncoderCountWheelRight : UDINT
SET
END_SET
END_PROPERTY

{attribute 'monitoring' := 'call'}
PROPERTY SetPointSpeedLeft : REAL
GET
END_GET
END_PROPERTY

{attribute 'monitoring' := 'call'}
PROPERTY SetPointSpeedRight : REAL
GET
END_GET
END_PROPERTY

END_INTERFACE

// ---- Components/Navitrol/Interface/I_Navitrol_GoToDestination.TcIO
INTERFACE I_Navitrol_GoToDestination EXTENDS I_Base

METHOD Execute : BOOL;
VAR_INPUT
	DestinationID : UDINT;
END_VAR
END_METHOD

{attribute 'monitoring' := 'call'}
PROPERTY Result : UDINT
GET
END_GET
END_PROPERTY

END_INTERFACE

// ---- Components/Navitrol/Interface/I_Navitrol_InitializePosition.TcIO
INTERFACE I_Navitrol_InitializePosition EXTENDS I_Base

METHOD InitializePosition : BOOL
VAR_INPUT
	X	  : REAL;	   //		X - map coordinate OF the AGV in meters
	Y	  : REAL;	   //		Y - map coordinate of the AGV in meters
	H	  : REAL := 0; //		Heading of the AGV on the map in radians
	Level : DINT := 0; //	The level ID on which the AGV is located
END_VAR
END_METHOD

END_INTERFACE

// ---- Components/Navitrol/Interface/I_Navitrol_OmniDriveMotorControl.TcIO
INTERFACE I_Navitrol_OmniDriveMotorControl EXTENDS I_Base

END_INTERFACE

// ---- Components/Navitrol/Interface/I_Navitrol_ReturnToRoute.TcIO
INTERFACE I_Navitrol_ReturnToRoute EXTENDS I_Base

METHOD Execute : BOOL
END_METHOD

END_INTERFACE

// ---- Components/Navitrol/Interface/I_Navitrol_Status.TcIO
INTERFACE I_Navitrol_Status EXTENDS I_Base

PROPERTY NavitrolStatus : REFERENCE TO ST_3102_Navitrol_status
GET
END_GET
END_PROPERTY

PROPERTY SupervisorStatus : REFERENCE TO ST_3002_Supervisor_Status
GET
END_GET
END_PROPERTY

END_INTERFACE

// ---- Components/Navitrol/Interface/I_Navitrol_StreamVelocity.TcIO
INTERFACE I_Navitrol_StreamVelocity EXTENDS I_Base, I_Enablable, I_TaskResult

METHOD SetTargetVelocity
VAR_INPUT
	TargetVelocity : LREAL; // Desired velocity setpoint (signed)
END_VAR
END_METHOD

END_INTERFACE

// ---- MAIN.TcPOU
PROGRAM MAIN
VAR
	Simulated				   : BOOL := FALSE;
	AmrModule				   : AmrModule('AMR Module');
	MachineHmiTree			   : GetSystemTreeJsonHmiVisitor<1000>('MAIN');
	SetSafetySimulationVisitor : SetSafetySimulationVisitor;
END_VAR

_AppInfo.KeepOutputsOnBP := TRUE;
IF NOT AmrModule.Initialized THEN
	AmrModule.Initialize();
	MachineHmiTree.GetTree(AmrModule);
	//
	IF Simulated THEN
		SetSafetySimulationVisitor.Diag	 := 0;
		SetSafetySimulationVisitor.State := 1;
		AmrModule.Components.Accept(SetSafetySimulationVisitor);
	END_IF

	RETURN;
END_IF

AmrModule.CyclicLogic();

END_PROGRAM

// ---- AMR/AmrModule.TcPOU
FUNCTION_BLOCK AmrModule EXTENDS PackMLModule IMPLEMENTS I_AmrModule
VAR
	Events			  : TcEventClass('AMR Module');
	EventReactor	  : EventReactorPackMLVisitor('Event Reaction', THIS^);
	SyncedSquareWaves : SyncedSquareWaves('Waves');

	//
	Navitrol_TcpIpConnection				   : TcpIpConnection('Navitrol Connection');
	Navitrol_Status							   : Msg3002_NavitrolStatus('Navitrol Status', Navitrol_TcpIpConnection); // Send AMR status and recieve Navitrol status
	Navitrol_InitializePosition				   : Msg1001_InitializePosition('Navitrol Initialize Position', Navitrol_TcpIpConnection);
	Navitrol_MeasurmentUpdateDifferentialDrive : Msg1016_MeasurmentUpdateDifferentialDrive('Navitrol Drive Control', Navitrol_TcpIpConnection);
	Navitrol_GoToDestination				   : Msg3005_GoToDestination('Navitrol Go To Destination', Navitrol_TcpIpConnection);
	Navitrol_ReturnToRoute					   : Msg3024_ReturnToRoute('Navitrol return to route', Navitrol_TcpIpConnection);
	Navitrol_StopHoldRelease				   : Msg3001_HoldRelease('Navitrol release hold', Navitrol_TcpIpConnection);

	// Wheel Left
	WheelLeftRef			  : AXIS_REF;
	_WheelLeft				  : AxisPTP('Wheel Left', WheelLeftRef);
	WheelLeft_HMI			  : AxisPTP_HMI('Wheel Left', _WheelLeft, '°');
	WheelLeft_TcEvents		  : Axis_TcEvents('Wheel Left', _WheelLeft);
	_WheelLeft_StreamVelocity : Navitrol_StreamVelocity('Velocity Stream Wheel Left', WheelLeftRef);

	// Wheel Right
	WheelRightRef			   : AXIS_REF;
	_WheelRight				   : AxisPTP('Wheel Right', WheelRightRef);
	WheelRight_HMI			   : AxisPTP_HMI('Wheel Right', _WheelRight, '°');
	WheelRight_TcEvents		   : Axis_TcEvents('Wheel Right', _WheelRight);
	_WheelRight_StreamVelocity : Navitrol_StreamVelocity('Velocity Stream Wheel Right', WheelRightRef);

	//
	EncoderSpeedIn AT %I*	 : INT;
	EncoderSpeed			 : AnalogInput('Encoder Speed', EncoderSpeedIn);
	EncoderPositionIn AT %I* : INT;
	EncoderPosition			 : AnalogInput('Encoder Position', EncoderPositionIn);
	Encoder_HMI				 : Encoder_HMI('Mouser DHK Encoder', EncoderSpeed, EncoderPosition);

	// Safety
	SafetyResetELM		 : SafetyResetPulse('Safety Reset');
	SafetyGroupReset	 : SafetyResetPulse('Safety Reset');
	SafetyInputGroup	 : SafetyGroup_TcEvents('Safety Input Group')	   := (ResetFunction := SafetyGroupReset, AutoResetFaults := TRUE);
	SafetyMotionGroup	 : SafetyGroup_TcEvents('Safety Motion Group')	   := (ResetFunction := SafetyGroupReset, AutoResetFaults := TRUE);
	SafetyLiftSpeedGroup : SafetyGroup_TcEvents('Safety Lift Speed Group') := (ResetFunction := SafetyGroupReset, AutoResetFaults := TRUE);
	SafetyReset			 : SafetyResetPulse('Safety Reset');
	SafetyEstop			 : SafetyEstopFB_TcEvents('E-Stop')		  := (ResetFunction := SafetyReset, SafetyGroup := SafetyInputGroup);
	SafetyScannerLeuze	 : SafetyMonFB_TcEvents('Leuze Scanner')  := (ActiveAlarm := TRUE, SafetyGroup := SafetyInputGroup, ActiveName := 'obstructed!');
	SafetyScannerHokuyo	 : SafetyMonFB_TcEvents('Hokuyo Scanner') := (ActiveAlarm := TRUE, SafetyGroup := SafetyInputGroup, ActiveName := 'obstructed!');

	// EP
	EP3751_IO AT %I*		 : ST_EP3751;
	EP3751_Accelerometer_HMI : EP3751_Accelerometer_HMI('EP3751 - Gyro', EP3751_IO);
END_VAR

VAR
	(* PackML State Statemachine     
        Aborting    = Transition to error state        
        Aborted     = Error State or Started
        Clearing    = Error Reset
        Stopped     = Idle, no error, manual operation of devices
        Stopping    = Stop transition to Stopped
        Starting    = Start System in Automatic
        Execute     = Running & Stream Velocity
        Suspending  = Stop AMR due to Safety Scanner
        Suspended   = Wait for Safety Scanner OK
        Unsuspending= Resume movement            
    *)
END_VAR

VAR
	AmrModule_HMI		   : AmrModule_HMI('AMR Module', _Statemachine, THIS^);
	_BypassScanners AT %Q* : BOOL;
	Navitrol_HMI		   : Navitrol_HMI('Navitrol', Navitrol_Status, Navitrol_TcpIpConnection);
END_VAR

VAR PERSISTENT
	{ attribute 'TcHmiSymbol.AddSymbol' }
	{ attribute 'TcHmiSymbol.AddSymbol.UserGroups' := '__SystemAdministrators, Admin' }
	Recipe_HMI : ST_Recipe;
END_VAR

VAR
	_Override		: LREAL := 100.0;
	Destination		: UDINT;
	COEDriveControl : COEDriveControl;
END_VAR

METHOD Aborted : BOOL;
END_METHOD

METHOD Aborting  : BOOL;
CASE SequenceState OF
	0:
		_WheelLeft_StreamVelocity.Disable();
		_WheelRight_StreamVelocity.Disable();
		_WheelLeft.Stop();
		_WheelRight.Stop();
		COEDriveControl.Enable := FALSE;
		NextMinorStep(SequenceState);

	1:
		IF NOT _WheelLeft.Busy AND NOT _WheelRight.Busy THEN
			NextStep(SequenceState);
		END_IF

	10:
		_WheelLeft.Disable();
		_WheelRight.Disable();
		NextStep(SequenceState);

	20:
		Aborting := TRUE;
END_CASE
END_METHOD

METHOD AmrEvents
IF NOT SafetyEstop.OK THEN
	Navitrol_Status.SupervisorStatus.Set_Estop := E_3002_Set_ESTOP.Set_ESTOP;
END_IF

IF Navitrol_TcpIpConnection.ConnectionState <> E_SocketConnectionState.eSOCKET_CONNECTED THEN
	IF Statemachine.Mode.CurrentMode <> E_PMLProtectedUnitMode.Manual THEN
		Events.RaiseEvent(E_AmrModule.NavitrolComError);
	END_IF
END_IF
END_METHOD

PROPERTY BypassScanners : BOOL
SET
_BypassScanners := BypassScanners;
END_SET
END_PROPERTY

METHOD Clearing : BOOL;
VAR_INST
	SafetyResetTon : TON;
END_VAR
CASE SequenceState OF
	0:
		ResetSafety();
		NextStep(SequenceState);
		COEDriveControl.Reset := TRUE;
		SafetyResetTon(IN := FALSE);

	10: // Wait for Safety signal propagation to drives
		SafetyResetTon(IN := TRUE, PT := T#200MS);
		IF SafetyResetTon.Q THEN
			SafetyResetELM.Execute();
			NextMinorStep(SequenceState);
		END_IF

	11:
		IF NOT SafetyResetELM.Busy THEN
			NextStep(SequenceState);
		END_IF

	20:
		ResetComponents(); // Call Reset on every component implementing I_Resettable
		COEDriveControl.Reset := FALSE;
		NextStep(SequenceState);

	30:
		Navitrol_Status.SupervisorStatus.Set_Estop := E_3002_Set_ESTOP.Release_ESTOP;
		Clearing								   := TRUE;
END_CASE
END_METHOD

METHOD Execute : BOOL;
VAR_INST
	WaitTime : TON;
END_VAR
IF (NOT SafetyScannerLeuze.OK OR NOT SafetyScannerHokuyo.OK) AND NOT _BypassScanners THEN
	Statemachine.ChangeState(E_PmlCommand.Suspend);
	RETURN;
END_IF

CASE SequenceState OF
	0:
		WaitTime(IN := FALSE);
		IF Navitrol_Status.NavitrolStatus.State = E_3102_State.HOLD_STATE THEN
			SequenceState := 11;
		ELSIF Navitrol_Status.NavitrolStatus.State = E_3102_State.AUTO_STATE THEN
			SequenceState := 11;
		ELSE
			NextStep(SequenceState);
		END_IF

	10:
		IF Navitrol_GoToDestination.Execute(Destination) THEN
			NextMinorStep(SequenceState);
		END_IF

	11:
		IF Navitrol_Status.NavitrolStatus.State = E_3102_State.HOLD_STATE THEN
			IF Destination = 4 THEN
				Destination := 1;
			ELSE
				Destination := Destination + 1;
			END_IF

			WaitTime(IN := FALSE);
			NextStep(SequenceState);
		END_IF

		// Route ended - simulation route
		WaitTime(IN := TRUE, PT := T#1S);
		IF WaitTime.Q THEN
			WaitTime(IN := FALSE);
			IF Navitrol_Status.NavitrolStatus.State = E_3102_State.STANDBY_STATE THEN
				SequenceState := 0;
			END_IF
		END_IF

	20:
		COEDriveControl.SetVelIncr := 50;
		COEDriveControl.Enable	   := TRUE;
		NextMinorStep(SequenceState);

	21:
		IF EncoderPositionIn >= 20_000 THEN
			COEDriveControl.Enable := FALSE;
			NextStep(SequenceState);
		END_IF

	30:
		WaitTime(IN := TRUE, PT := T#2S);
		IF WaitTime.Q THEN
			WaitTime(IN := FALSE);
			NextStep(SequenceState);
		END_IF

	40:
		COEDriveControl.SetVelIncr := -50;
		COEDriveControl.Enable	   := TRUE;
		NextMinorStep(SequenceState);

	41:
		IF EncoderPositionIn <= -20_000 THEN
			COEDriveControl.Enable := FALSE;
			NextStep(SequenceState);
		END_IF

	50:
		IF Navitrol_StopHoldRelease.Execute() THEN
			NextMinorStep(SequenceState);
		END_IF

	51:
		IF Navitrol_Status.NavitrolStatus.State = E_3102_State.AUTO_STATE THEN
			WaitTime(IN := FALSE);
			SequenceState := 11;
		END_IF

		// Route ended - simulation route
		WaitTime(IN := TRUE, PT := T#1S);
		IF WaitTime.Q THEN
			WaitTime(IN := FALSE);
			IF Navitrol_Status.NavitrolStatus.State = E_3102_State.STANDBY_STATE THEN
				SequenceState := 0;
			END_IF

			IF Navitrol_Status.NavitrolStatus.State = E_3102_State.HOLD_STATE THEN
				SequenceState := 50;
			END_IF
		END_IF
END_CASE
END_METHOD

(*FB_Init is always available implicitly and it is used primarily for initialization.
The return value is not evaluated. For a specific influence, you can also declare the
methods explicitly and provide additional code there with the standard initialization
code. You can evaluate the return value.*)
METHOD FB_Init : BOOL
VAR_INPUT
	(* TRUE: the retain variables are initialized (reset warm / reset cold)*)
	bInitRetains : BOOL;

	(* TRUE: the instance will be copied to the copy code afterward (online change)   *)
	bInCopyCode : BOOL;
	Name		: Core.T_MaxString;
END_VAR
Events.GenerateTcEvents(Name, ADR(TC_Events.AmrModule), SIZEOF(ST_AmrModule));
Events.RegisterWithParent(THIS^);
EventReactor.RegisterWithParent(THIS^);
AmrModule_HMI.RegisterWithParent(THIS^);
SyncedSquareWaves.RegisterWithParent(THIS^);
_Statemachine.RegisterWithParent(THIS^);
_Statemachine.Name := _Name;

//
Navitrol_TcpIpConnection.IP				  := '127.0.0.1';
Navitrol_TcpIpConnection.PollTime		  := T#1MS;
Navitrol_TcpIpConnection.Port			  := 2000;
Navitrol_TcpIpConnection.ReceiveTimeout	  := T#10S;
Navitrol_TcpIpConnection.ReconnectionTime := T#10S;
Navitrol_TcpIpConnection.SendInterval	  := T#1MS;
Navitrol_TcpIpConnection.RegisterWithParent(THIS^);
Navitrol_Status.RegisterWithParent(THIS^);
Navitrol_InitializePosition.RegisterWithParent(THIS^);
Navitrol_MeasurmentUpdateDifferentialDrive.RegisterWithParent(THIS^);
Navitrol_HMI.RegisterWithParent(THIS^);
Navitrol_GoToDestination.RegisterWithParent(THIS^);
Navitrol_ReturnToRoute.RegisterWithParent(THIS^);
Navitrol_StopHoldRelease.RegisterWithParent(THIS^);

//
_WheelLeft.RegisterWithParent(THIS^);
WheelLeft_HMI.RegisterWithParent(THIS^);
WheelLeft_TcEvents.RegisterWithParent(THIS^);
_WheelLeft_StreamVelocity.RegisterWithParent(THIS^);

//
_WheelRight.RegisterWithParent(THIS^);
WheelRight_HMI.RegisterWithParent(THIS^);
WheelRight_TcEvents.RegisterWithParent(THIS^);
_WheelRight_StreamVelocity.RegisterWithParent(THIS^);

//
SafetyInputGroup.RegisterWithParent(THIS^);
SafetyLiftSpeedGroup.RegisterWithParent(THIS^);
SafetyMotionGroup.RegisterWithParent(THIS^);
SafetyEstop.RegisterWithParent(THIS^);
SafetyScannerLeuze.RegisterWithParent(THIS^);
SafetyScannerHokuyo.RegisterWithParent(THIS^);
SafetyScannerLeuze.SetEventReactions(0,
									 0,
									 0,
									 0,
									 0);

SafetyScannerHokuyo.SetEventReactions(0,
									  0,
									  0,
									  0,
									  0);

SafetyResetELM.RegisterWithParent(THIS^);

//
EncoderSpeed.RegisterWithParent(THIS^);
EncoderPosition.RegisterWithParent(THIS^);
Encoder_HMI.RegisterWithParent(THIS^);

//
EP3751_Accelerometer_HMI.RegisterWithParent(THIS^);
END_METHOD

(* This Module will be done initializeing when ModuleInitialized := TRUE;, subequently all subitems will be called to be initialized*)
METHOD Initializing
VAR_INST
	UnitModeConfig : FB_PMLUnitModeConfig;
	SequenceState  : UDINT;
END_VAR
CASE SequenceState OF
	0:
		UnitModeConfig(eMode						  := E_PMLProtectedUnitMode.Production,
					   sName						  := 'Production',
					   bDisableClearing				  := FALSE,
					   bDisableStarting				  := FALSE,
					   bDisableSuspended			  := FALSE,
					   bDisableStopping				  := FALSE,
					   bDisableAborting				  := FALSE,
					   bDisableHolding				  := TRUE,
					   bDisableHeld					  := TRUE,
					   bDisableUnholding			  := TRUE,
					   bDisableSuspending			  := FALSE,
					   bDisableUnsuspending			  := FALSE,
					   bDisableResetting			  := TRUE,
					   bDisableIdle					  := TRUE,
					   bDisableCompleting			  := TRUE,
					   bDisableComplete				  := TRUE,
					   bEnableUnitModeChangeStopped	  := TRUE,
					   bEnableUnitModeChangeIdle	  := FALSE,
					   bEnableUnitModeChangeSuspended := FALSE,
					   bEnableUnitModeChangeExecute	  := FALSE,
					   bEnableUnitModeChangeAborted	  := TRUE,
					   bEnableUnitModeChangeHeld	  := FALSE,
					   bEnableUnitModeChangeComplete  := FALSE,
					   bError						  =>,
					   nErrorId						  =>);

		UnitModeConfig(eMode						  := E_PMLProtectedUnitMode.Manual,
					   sName						  := 'Manual',
					   bDisableClearing				  := FALSE,
					   bDisableStarting				  := FALSE,
					   bDisableSuspended			  := TRUE,
					   bDisableStopping				  := FALSE,
					   bDisableAborting				  := FALSE,
					   bDisableHolding				  := TRUE,
					   bDisableHeld					  := TRUE,
					   bDisableUnholding			  := TRUE,
					   bDisableSuspending			  := TRUE,
					   bDisableUnsuspending			  := TRUE,
					   bDisableResetting			  := TRUE,
					   bDisableIdle					  := TRUE,
					   bDisableCompleting			  := TRUE,
					   bDisableComplete				  := TRUE,
					   bEnableUnitModeChangeStopped	  := TRUE,
					   bEnableUnitModeChangeIdle	  := FALSE,
					   bEnableUnitModeChangeSuspended := FALSE,
					   bEnableUnitModeChangeExecute	  := FALSE,
					   bEnableUnitModeChangeAborted	  := TRUE,
					   bEnableUnitModeChangeHeld	  := FALSE,
					   bEnableUnitModeChangeComplete  := FALSE,
					   bError						  =>,
					   nErrorId						  =>);

		SequenceState := SequenceState + 10;

	10:
		ModuleInitialized := TRUE;
END_CASE
END_METHOD

METHOD OnCyclicCall
VAR_INST
	HmiEnableDisable : HmiEnableDisableAllVisitor;
	SetOverride		 : SetAllOverrideVisitor;
	ProductionRT	 : R_TRIG;
	AutoResetTon	 : TON;
END_VAR
ProductionRT(CLK := _Statemachine.Mode.CurrentMode = E_PMLProtectedUnitMode.Production);
IF _Statemachine.Mode.CurrentMode = E_PMLProtectedUnitMode.Manual THEN
	HmiEnableDisable.EnableHmi(THIS^);
	IF Navitrol_HMI.NavitrolHasControl THEN
		_WheelLeft_StreamVelocity.Enable();
		_WheelRight_StreamVelocity.Enable();
	ELSE
		_WheelLeft_StreamVelocity.Disable();
		_WheelRight_StreamVelocity.Disable();
	END_IF
ELSE
	HmiEnableDisable.DisableHmi(THIS^);
	AmrModule_HMI.Enable();
	IF ProductionRT.Q THEN
		_WheelLeft_StreamVelocity.Disable();
		_WheelRight_StreamVelocity.Disable();
	END_IF
END_IF

IF (_Statemachine.CurrentState = E_PMLState.Aborted) OR (_Statemachine.CurrentState = E_PMLState.Stopped) THEN
	AutoResetTon(IN := NOT AutoResetTon.Q, PT := T#1S);
	IF AutoResetTon.Q THEN
		SafetyScannerLeuze.Reset();
		SafetyScannerHokuyo.Reset();
	END_IF;
END_IF

//
SetOverride.Set(THIS^, _Override);
AmrEvents();

//
EncoderPosition.Scale.InputMaximum	:= Encoder_HMI.Config.Position_InputMaximum;
EncoderPosition.Scale.InputMinimum	:= Encoder_HMI.Config.Position_InputMinimum;
EncoderPosition.Scale.OutputMaximum := Encoder_HMI.Config.Position_OutputMaximum;
EncoderPosition.Scale.OutputMinimum := Encoder_HMI.Config.Position_OutputMinimum;
EncoderSpeed.Scale.InputMaximum		:= Encoder_HMI.Config.Speed_InputMaximum;
EncoderSpeed.Scale.InputMinimum		:= Encoder_HMI.Config.Speed_InputMinimum;
EncoderSpeed.Scale.OutputMaximum	:= Encoder_HMI.Config.Speed_OutputMaximum;
EncoderSpeed.Scale.OutputMinimum	:= Encoder_HMI.Config.Speed_OutputMinimum;

//
COEDriveControl(Manual := (_Statemachine.Mode.CurrentMode = E_PMLProtectedUnitMode.Manual));

// (Diameter Wheel * 360deg)
Navitrol_MeasurmentUpdateDifferentialDrive.EncoderCountWheelLeft  := TO_UDINT(_WheelLeft.ActualPosition * 1_000);
Navitrol_MeasurmentUpdateDifferentialDrive.EncoderCountWheelRight := TO_UDINT(_WheelRight.ActualPosition * 1_000);
_WheelLeft_StreamVelocity.SetTargetVelocity(((360 * Navitrol_MeasurmentUpdateDifferentialDrive.SetPointSpeedLeft) / (PI * AMR_CONSTANT.WHEEL_DIAMETER)));
_WheelRight_StreamVelocity.SetTargetVelocity(((360 * Navitrol_MeasurmentUpdateDifferentialDrive.SetPointSpeedRight) / (PI * AMR_CONSTANT.WHEEL_DIAMETER)));
END_METHOD

{attribute 'monitoring' := 'call'}
PROPERTY Override : LREAL
SET
_Override := Override;

//SetOverrideVisitor.SetOverride(THIS^, _Override);
END_SET
END_PROPERTY

METHOD ResetSafety
SafetyEstop.Reset();
SafetyScannerLeuze.Reset();
SafetyScannerHokuyo.Reset();
END_METHOD

METHOD Starting  : BOOL;
CASE SequenceState OF
	0:
		IF Navitrol_InitializePosition.InitializePosition(21.23,
														  36.92,
														  TO_REAL(DEGREE_TO_RADIAN(90)),
														  0) THEN
			Destination := 1;
			NextMinorStep(SequenceState);
		END_IF

	1:
		IF Navitrol_Status.NavitrolStatus.State = E_3102_State.STANDBY_STATE OR Navitrol_Status.NavitrolStatus.State = E_3102_State.HOLD_STATE OR Navitrol_Status.NavitrolStatus.State = E_3102_State.AUTO_STATE THEN
			NextStep(SequenceState);
		END_IF

	10:
		_WheelLeft.Enable();
		_WheelRight.Enable();
		IF _WheelLeft.Enabled AND _WheelRight.Enabled THEN
			NextStep(SequenceState);
		END_IF

	20:
		_WheelLeft_StreamVelocity.Enable();
		_WheelRight_StreamVelocity.Enable();
		IF _WheelLeft_StreamVelocity.Enabled AND _WheelRight_StreamVelocity.Enabled THEN
			NextStep(SequenceState);
		END_IF

	30:
		Starting := TRUE;
END_CASE
END_METHOD

PROPERTY Statemachine : I_Statemachine
GET
Statemachine := _Statemachine;
END_GET
END_PROPERTY

METHOD Stopped  : BOOL;
END_METHOD

METHOD Stopping  : BOOL;
CASE SequenceState OF
	0: // Wait AMR not moving
		IF Navitrol_MeasurmentUpdateDifferentialDrive.SetPointSpeedLeft = 0.0 AND Navitrol_MeasurmentUpdateDifferentialDrive.SetPointSpeedRight = 0.0 THEN
			IF CompareLREAL(_WheelLeft.ActualVelocity, 0.0, 0.01) AND CompareLREAL(_WheelRight.ActualVelocity, 0.0, 0.01) THEN
				_WheelLeft_StreamVelocity.Disable();
				_WheelRight_StreamVelocity.Disable();
				_WheelLeft.Stop();
				_WheelRight.Stop();
				NextMinorStep(SequenceState);
			END_IF
		END_IF

	1:
		IF NOT _WheelLeft.Busy AND NOT _WheelRight.Busy THEN
			NextStep(SequenceState);
		END_IF

	10:
		_WheelLeft.Disable();
		_WheelRight.Disable();
		IF NOT _WheelLeft.Enabled AND NOT _WheelRight.Enabled THEN
			NextStep(SequenceState);
		END_IF

	20:
		Stopping := TRUE;
END_CASE
END_METHOD

METHOD Suspended : BOOL
IF SafetyScannerLeuze.OK AND SafetyScannerHokuyo.OK THEN
	Statemachine.ChangeState(E_PmlCommand.Unsuspend);
	RETURN;
END_IF
END_METHOD

METHOD Suspending : BOOL
CASE SequenceState OF
	0:
		Navitrol_Status.SupervisorStatus.Set_Estop := E_3002_Set_ESTOP.Set_ESTOP;
		_WheelLeft_StreamVelocity.Disable();
		_WheelRight_StreamVelocity.Disable();
        _WheelLeft.Stop();
		_WheelRight.Stop();
		NextMinorStep(SequenceState);

	1:
		IF  NOT _WheelLeft.Busy AND NOT _WheelRight.Busy THEN
			IF CompareLREAL(_WheelLeft.ActualVelocity, 0.0, 0.01) AND CompareLREAL(_WheelRight.ActualVelocity, 0.0, 0.01) THEN
				NextStep(SequenceState);
			END_IF
		END_IF

	10:
		_WheelLeft.Disable();
		_WheelRight.Disable();
		IF NOT _WheelLeft.Enabled AND NOT _WheelRight.Enabled THEN
			NextStep(SequenceState);
		END_IF

	20:
		Suspending := TRUE;
END_CASE
END_METHOD

METHOD Unsuspending : BOOL
VAR_INST
	SafetyResetTon : TON;
END_VAR
CASE SequenceState OF
	0:
		SafetyScannerLeuze.Reset();
		SafetyScannerHokuyo.Reset();
		NextMinorStep(SequenceState);

	1: // Wait for Safety signal propagation to drives
		SafetyResetTon(IN := TRUE, PT := T#200MS);
		IF SafetyResetTon.Q THEN
			SafetyResetELM.Execute();
			NextMinorStep(SequenceState);
		END_IF

	2:
		IF NOT SafetyResetELM.Busy THEN
			NextMinorStep(SequenceState);
		END_IF

	3:
		_WheelLeft.Enable();
		_WheelRight.Enable();
		_WheelLeft_StreamVelocity.Enable();
		_WheelRight_StreamVelocity.Enable();
		IF _WheelLeft.Enabled AND _WheelRight.Enabled THEN
			NextStep(SequenceState);
		END_IF

	10:
		Navitrol_Status.SupervisorStatus.Set_Estop := E_3002_Set_ESTOP.Release_ESTOP;
		NextStep(SequenceState);

	20:
		NextStep(SequenceState);

	30:
		IF Navitrol_GoToDestination.Execute(Destination) THEN
			Unsuspending := TRUE;
		END_IF
END_CASE
END_METHOD

PROPERTY WheelLeft : I_Axis_PTP
GET
WheelLeft := _WheelLeft;
END_GET
END_PROPERTY

PROPERTY WheelLeftStreamVelocity : I_Navitrol_StreamVelocity
GET
WheelLeftStreamVelocity := _WheelLeft_StreamVelocity;
END_GET
END_PROPERTY

PROPERTY WheelRight : I_Axis_PTP
GET
WheelRight := _WheelRight;
END_GET
END_PROPERTY

PROPERTY WheelRightStreamVelocity : I_Navitrol_StreamVelocity
GET
WheelRightStreamVelocity := _WheelRight_StreamVelocity;
END_GET
END_PROPERTY

END_FUNCTION_BLOCK

// ---- Components/Navitrol/Msg3002_NavitrolStatus.TcPOU
FUNCTION_BLOCK Msg3002_NavitrolStatus EXTENDS TcpIpCommandResultFilter IMPLEMENTS I_Navitrol_Status
VAR
	CycleTime		  : TIME := T#100MS; //maximum interval 1 second
	Timer			  : TON;
	Command			  : ST_TcpIpPayload;
	ReceiveBuffer	  : U_Recived_bytes_from_Navitrol;
	Supervisor_Status : ST_3002_Supervisor_Status;
	Navitrol_status	  : ST_3102_Navitrol_status;
END_VAR

METHOD CyclicLogic
SUPER^.CyclicLogic();
Timer(IN := NOT Timer.Q, PT := CycleTime);
IF Timer.Q AND TcpIpConnection.ConnectionState = eSOCKET_CONNECTED THEN
	F_SetHeaderInfo(Supervisor_Status);
	F_SetSectionHeaderInfo(Supervisor_Status.Manual_section);
	F_SetSectionHeaderInfo(Supervisor_Status.Battery_section);
	MEMSET(ADR(Command), 0, SIZEOF(Command));
	Command.Size := SIZEOF(Supervisor_Status);
	MEMCPY(ADR(Command.Data), ADR(Supervisor_Status), Command.Size);
	TcpIpConnection.SendCommand(ADR(Command));
	CommandActive := TRUE;
END_IF
END_METHOD

PROPERTY NavitrolStatus : REFERENCE TO ST_3102_Navitrol_status
GET
NavitrolStatus REF= Navitrol_status;
END_GET
END_PROPERTY

PROPERTY SupervisorStatus : REFERENCE TO ST_3002_Supervisor_Status
GET
SupervisorStatus REF= Supervisor_Status;
END_GET
END_PROPERTY

METHOD UpdateCommandResult
VAR_INPUT
	Response : POINTER TO ST_TcpIpPayload;
END_VAR

VAR_INST
	ReceiveCounter : UDINT;
END_VAR
MEMCPY(ADR(ReceiveBuffer), ADR(Response^.Data), SIZEOF(ReceiveBuffer));
IF ReceiveBuffer.Header.Message_ID = 3102 THEN
	ReceiveCounter := ReceiveCounter + 1;
	MEMCPY(destAddr := ADR(Navitrol_status), srcAddr := ADR(ReceiveBuffer), n := SIZEOF(Navitrol_status));
	CommandActive := FALSE;
END_IF
END_METHOD

END_FUNCTION_BLOCK

// ---- Components/Navitrol/Supervisor to Navitrol message/F_SetHeaderInfo.TcPOU
//Use this to populate "ST_SupervisorHeader" in the message being sent from Supervisor to Navitrol
FUNCTION F_SetHeaderInfo : HRESULT;
VAR_INPUT
	Msg : ANY;
END_VAR

VAR
	MsgHeader			  : ST_SupervisorHeader;
	JsonDataType		  : FB_JsonReadWriteDataType;
	DataTypeName		  : STRING;
	Message_ID			  : UINT;
	GetDataTypeNameResult : HRESULT;
	i					  : INT;
	StartPos			  : INT;
	EndPos				  : INT;
	IDString			  : STRING;
	ParseSuccess		  : BOOL;
END_VAR

IF Msg.diSize < 0 THEN
	F_SetHeaderInfo := S_FALSE;
	RETURN;
END_IF

DataTypeName := JsonDataType.GetDataTypeNameByAddress(nData := TO_UDINT(Msg.diSize), pData := Msg.pValue, hrErrorCode => GetDataTypeNameResult);

// Parse Message_ID from DataTypeName (e.g., 'ST_3002_Supervisor_Status' -> 3002)
ParseSuccess := FALSE;
StartPos	 := FIND(DataTypeName, 'ST_');
IF StartPos > 0 THEN
	StartPos := StartPos + 3; // Move past 'ST_'

	// Find the next underscore after the ID
	EndPos := 0;
	FOR i := StartPos TO LEN(DataTypeName) DO
		IF MID(DataTypeName, 1, i) = '_' THEN
			EndPos := i;
			EXIT;
		END_IF
	END_FOR

	IF EndPos > StartPos THEN
		// Extract the ID substring
		IDString	 := MID(DataTypeName, EndPos - StartPos, StartPos);
		Message_ID	 := STRING_TO_UINT(IDString);
		ParseSuccess := TRUE;
	END_IF
END_IF

// Fallback if parsing fails
IF NOT ParseSuccess THEN
	Message_ID		:= 0;
	F_SetHeaderInfo := S_FALSE;
	RETURN;
END_IF

// All messages start with ST_SupervisorHeader
MsgHeader.Protocol_version := 4;
MsgHeader.Message_ID	   := Message_ID;
MsgHeader.Message_length   := TO_UDINT(Msg.diSize);

// Copy populated header into Msg
MEMCPY(destAddr := Msg.pValue, srcAddr := ADR(MsgHeader), n := SIZEOF(MsgHeader));
F_SetHeaderInfo := S_OK;

END_FUNCTION

// ---- Components/Navitrol/Supervisor to Navitrol message/3002/Components/Sections/F_SetSectionHeaderInfo.TcPOU
FUNCTION F_SetSectionHeaderInfo : HRESULT
VAR_INPUT
	Section : ANY;
END_VAR

VAR
	SectionHeader		  : ST_SectionHeader;
	JsonDataType		  : FB_JsonReadWriteDataType;
	DataTypeName		  : STRING;
	Message_ID			  : UINT;
	GetDataTypeNameResult : HRESULT;
	i					  : INT;
	StartPos			  : INT;
	EndPos				  : INT;
	IDString			  : STRING;
	ParseSuccess		  : BOOL;
END_VAR

IF Section.diSize < 0 THEN
	F_SetSectionHeaderInfo := S_FALSE;
	RETURN;
END_IF

DataTypeName := JsonDataType.GetDataTypeNameByAddress(nData := TO_UDINT(Section.diSize), pData := Section.pValue, hrErrorCode => GetDataTypeNameResult);

// Parse Message_ID from DataTypeName (e.g., 'ST_3002_2_Manual_section' -> 2)
ParseSuccess := FALSE;
StartPos	 := FIND(DataTypeName, 'ST_3002_');
IF StartPos > 0 THEN
	StartPos := StartPos + 8; // Move past 'ST_3002_'

	// Find the next underscore after the ID
	EndPos := 0;
	FOR i := StartPos TO LEN(DataTypeName) DO
		IF MID(DataTypeName, 1, i) = '_' THEN
			EndPos := i;
			EXIT;
		END_IF
	END_FOR

	IF EndPos > StartPos THEN
		// Extract the ID substring
		IDString	 := MID(DataTypeName, EndPos - StartPos, StartPos);
		Message_ID	 := STRING_TO_UINT(IDString);
		ParseSuccess := TRUE;
	END_IF
END_IF

// Fallback if parsing fails
IF NOT ParseSuccess THEN
	Message_ID			   := 0;
	F_SetSectionHeaderInfo := S_FALSE;
	RETURN;
END_IF

// All 3002 messages sections start with ST_SectionHeader
SectionHeader.Section_ID	 := Message_ID;
SectionHeader.Section_length := TO_UDINT(Section.diSize);

// Copy populated header into Section
MEMCPY(destAddr := Section.pValue, srcAddr := ADR(SectionHeader), n := SIZEOF(SectionHeader));
F_SetSectionHeaderInfo := S_OK;

END_FUNCTION

// ---- Components/Navitrol/Msg1001_InitializePosition.TcPOU
FUNCTION_BLOCK Msg1001_InitializePosition EXTENDS TcpIpCommandResultFilter IMPLEMENTS I_Navitrol_InitializePosition
VAR
	Command							: ST_TcpIpPayload;
	ReceiveBuffer					: U_Recived_bytes_from_Navitrol;
	Position_initialization_started : ST_1100_Position_initialization_started;
	Position_initialized			: ST_1101_Position_initialized;
	Initialize_position				: ST_1001_Initialize_position := (X := 100.0, Y := 150.0);
END_VAR

METHOD InitializePosition : BOOL
VAR_INPUT
	X	  : REAL;	   //		X - map coordinate OF the AGV in meters
	Y	  : REAL;	   //		Y - map coordinate of the AGV in meters
	H	  : REAL := 0; //		Heading of the AGV on the map in radians
	Level : DINT := 0; //	The level ID on which the AGV is located
END_VAR
IF TcpIpConnection.ConnectionState = eSOCKET_CONNECTED THEN
	F_SetHeaderInfo(Initialize_position);
	MEMSET(ADR(Command), 0, SIZEOF(Command));
	Initialize_position.X	  := X;
	Initialize_position.Y	  := Y;
	Initialize_position.H	  := H;
	Initialize_position.Level := Level;

	//
	Command.Size := SIZEOF(Initialize_position);
	MEMCPY(ADR(Command.Data), ADR(Initialize_position), Command.Size);
	TcpIpConnection.SendCommand(ADR(Command));
	CommandActive	   := TRUE;
	InitializePosition := TRUE;
END_IF
END_METHOD

METHOD UpdateCommandResult
VAR_INPUT
	Response : POINTER TO ST_TcpIpPayload;
END_VAR

VAR_INST
	ReceiveCounter : UDINT;
END_VAR
MEMCPY(ADR(ReceiveBuffer), ADR(Response^.Data), SIZEOF(ReceiveBuffer));
IF ReceiveBuffer.Header.Message_ID = 1100 THEN
	ReceiveCounter := ReceiveCounter + 1;
	MEMCPY(destAddr := ADR(Position_initialization_started), srcAddr := ADR(ReceiveBuffer), n := SIZEOF(Position_initialization_started));
	CommandActive := FALSE;
END_IF

IF ReceiveBuffer.Header.Message_ID = 1101 THEN
	ReceiveCounter := ReceiveCounter + 1;
	MEMCPY(destAddr := ADR(Position_initialized), srcAddr := ADR(ReceiveBuffer), n := SIZEOF(Position_initialized));
	CommandActive := FALSE;
END_IF
END_METHOD

END_FUNCTION_BLOCK

// ---- Components/Navitrol/Msg1016_MeasurmentUpdateDifferentialDrive.TcPOU
FUNCTION_BLOCK Msg1016_MeasurmentUpdateDifferentialDrive EXTENDS TcpIpCommandResultFilter IMPLEMENTS I_Navitrol_DifferentialDriveMotorControl
VAR
	CycleTime							  : TIME := T#30MS; //This needs to match the Navitrol parameter "control_interval_us"
	Timer								  : TON;
	Command								  : ST_TcpIpPayload;
	ReceiveBuffer						  : U_Recived_bytes_from_Navitrol;
	Measurement_update_differential_drive : ST_1016_Measurement_update_differential_drive;
	Motor_Control_Differential			  : ST_1116_Motor_Control_Differential;
END_VAR

METHOD CyclicLogic
SUPER^.CyclicLogic();
Measurement_update_differential_drive.Timestamp := Measurement_update_differential_drive.Timestamp + TO_UINT(_Taskinfo[GETCURTASKINDEXEX()].CycleTime);
Timer(IN := NOT Timer.Q, PT := CycleTime);
IF Timer.Q AND TcpIpConnection.ConnectionState = eSOCKET_CONNECTED THEN
	F_SetHeaderInfo(Measurement_update_differential_drive);
	Measurement_update_differential_drive.Message_number := Measurement_update_differential_drive.Message_number + 1;

	//
	MEMSET(ADR(Command), 0, SIZEOF(Command));
	Command.Size := SIZEOF(Measurement_update_differential_drive);
	MEMCPY(ADR(Command.Data), ADR(Measurement_update_differential_drive), Command.Size);
	TcpIpConnection.SendPriorityCommand(ADR(Command));
	CommandActive := TRUE;
END_IF
END_METHOD

{attribute 'monitoring' := 'call'}
PROPERTY EncoderCountWheelLeft : UDINT
SET
Measurement_update_differential_drive.Odometry_left_wheel := EncoderCountWheelLeft;
END_SET
END_PROPERTY

{attribute 'monitoring' := 'call'}
PROPERTY EncoderCountWheelRight : UDINT
SET
Measurement_update_differential_drive.Odometry_right_wheel := EncoderCountWheelRight;
END_SET
END_PROPERTY

{attribute 'monitoring' := 'call'}
PROPERTY SetPointSpeedLeft : REAL
GET
SetPointSpeedLeft := Motor_Control_Differential.Speed_Left;
END_GET
END_PROPERTY

{attribute 'monitoring' := 'call'}
PROPERTY SetPointSpeedRight : REAL
GET
SetPointSpeedRight := Motor_Control_Differential.Speed_Right;
END_GET
END_PROPERTY

METHOD UpdateCommandResult
VAR_INPUT
	Response : POINTER TO ST_TcpIpPayload;
END_VAR

VAR_INST
	ReceiveCounter : UDINT;
END_VAR
MEMCPY(ADR(ReceiveBuffer), ADR(Response^.Data), SIZEOF(ReceiveBuffer));
IF ReceiveBuffer.Header.Message_ID = 1116 THEN
	ReceiveCounter := ReceiveCounter + 1;
	MEMCPY(destAddr := ADR(Motor_Control_Differential), srcAddr := ADR(ReceiveBuffer), n := SIZEOF(Motor_Control_Differential));
	CommandActive := FALSE;
END_IF
END_METHOD

END_FUNCTION_BLOCK

// ---- Components/Navitrol/Msg3005_GoToDestination.TcPOU
FUNCTION_BLOCK Msg3005_GoToDestination EXTENDS TcpIpCommandResultFilter IMPLEMENTS I_Navitrol_GoToDestination
VAR
	Command				  : ST_TcpIpPayload;
	ReceiveBuffer		  : U_Recived_bytes_from_Navitrol;
	GoToDestination		  : ST_3005_GoToDestination;
	GoToDestinationResult : ST_3105_GoToDestinationResult;
END_VAR

METHOD Execute : BOOL;
VAR_INPUT
	DestinationID : UDINT;
END_VAR
IF TcpIpConnection.ConnectionState = eSOCKET_CONNECTED THEN
	F_SetHeaderInfo(GoToDestination);
	MEMSET(ADR(Command), 0, SIZEOF(Command));
	GoToDestination.DestinationID := DestinationId;
	Command.Size				  := SIZEOF(GoToDestination);
	MEMCPY(ADR(Command.Data), ADR(GoToDestination), Command.Size);
	TcpIpConnection.SendCommand(ADR(Command));
	CommandActive := TRUE;
	Execute		  := TRUE;
END_IF
END_METHOD

{attribute 'monitoring' := 'call'}
PROPERTY Result : UDINT
GET
Result := GoToDestinationResult.GoToResult;
END_GET
END_PROPERTY

METHOD UpdateCommandResult
VAR_INPUT
	Response : POINTER TO ST_TcpIpPayload;
END_VAR

VAR_INST
	ReceiveCounter : UDINT;
END_VAR
MEMCPY(ADR(ReceiveBuffer), ADR(Response^.Data), SIZEOF(ReceiveBuffer));
IF ReceiveBuffer.Header.Message_ID = 3105 THEN
	ReceiveCounter := ReceiveCounter + 1;
	MEMCPY(destAddr := ADR(GoToDestinationResult), srcAddr := ADR(ReceiveBuffer), n := SIZEOF(GoToDestinationResult));
	CommandActive := FALSE;
END_IF
END_METHOD

END_FUNCTION_BLOCK

// ---- Components/Navitrol/Msg3024_ReturnToRoute.TcPOU
FUNCTION_BLOCK Msg3024_ReturnToRoute EXTENDS TcpIpCommandResultFilter IMPLEMENTS I_Navitrol_ReturnToRoute
VAR
	Command				: ST_TcpIpPayload;
	ReceiveBuffer		: U_Recived_bytes_from_Navitrol;
	ReturnToRoute		: ST_3024_ReturnToRoute;
	ReturnToRouteResult : ST_3124_ReturnToRouteResponse;
END_VAR

METHOD Execute : BOOL;
IF TcpIpConnection.ConnectionState = eSOCKET_CONNECTED THEN
	F_SetHeaderInfo(ReturnToRoute);
	MEMSET(ADR(Command), 0, SIZEOF(Command));
	Command.Size := SIZEOF(ReturnToRoute);
	MEMCPY(ADR(Command.Data), ADR(ReturnToRoute), Command.Size);
	TcpIpConnection.SendCommand(ADR(Command));
	CommandActive := TRUE;
	Execute		  := TRUE;
END_IF
END_METHOD

METHOD UpdateCommandResult
VAR_INPUT
	Response : POINTER TO ST_TcpIpPayload;
END_VAR

VAR_INST
	ReceiveCounter : UDINT;
END_VAR
MEMCPY(ADR(ReceiveBuffer), ADR(Response^.Data), SIZEOF(ReceiveBuffer));
IF ReceiveBuffer.Header.Message_ID = 3124 THEN
	ReceiveCounter := ReceiveCounter + 1;
	MEMCPY(destAddr := ADR(ReturnToRouteResult), srcAddr := ADR(ReceiveBuffer), n := SIZEOF(ReturnToRouteResult));
	CommandActive := FALSE;
END_IF
END_METHOD

END_FUNCTION_BLOCK

// ---- Components/Navitrol/Msg3001_HoldRelease.TcPOU
FUNCTION_BLOCK Msg3001_HoldRelease EXTENDS TcpIpCommandResultFilter IMPLEMENTS I_Navitrol_ReturnToRoute
VAR
	Command		  : ST_TcpIpPayload;
	ReceiveBuffer : U_Recived_bytes_from_Navitrol;
	ReleaseHold	  : ST_3001_ReleaseHoldState;
	HoldReleased  : ST_3101_HoldReleased;
END_VAR

METHOD Execute : BOOL
IF TcpIpConnection.ConnectionState = eSOCKET_CONNECTED THEN
	F_SetHeaderInfo(ReleaseHold);
	MEMSET(ADR(Command), 0, SIZEOF(Command));
	Command.Size := SIZEOF(ReleaseHold);
	MEMCPY(ADR(Command.Data), ADR(ReleaseHold), Command.Size);
	TcpIpConnection.SendCommand(ADR(Command));
	CommandActive := TRUE;
	Execute		  := TRUE;
END_IF
END_METHOD

METHOD UpdateCommandResult
VAR_INPUT
	Response : POINTER TO ST_TcpIpPayload;
END_VAR

VAR_INST
	ReceiveCounter : UDINT;
END_VAR
MEMCPY(ADR(ReceiveBuffer), ADR(Response^.Data), SIZEOF(ReceiveBuffer));
IF ReceiveBuffer.Header.Message_ID = 3101 THEN
	ReceiveCounter := ReceiveCounter + 1;
	MEMCPY(destAddr := ADR(HoldReleased), srcAddr := ADR(ReceiveBuffer), n := SIZEOF(HoldReleased));
	CommandActive := FALSE;
END_IF
END_METHOD

END_FUNCTION_BLOCK

// ---- Components/Navitrol/Navitrol_StreamVelocity.TcPOU
FUNCTION_BLOCK Navitrol_StreamVelocity EXTENDS CyclicComponent IMPLEMENTS I_Navitrol_StreamVelocity
VAR
	Axis			   : REFERENCE TO AXIS_REF;
	TargetVelocity	   : LREAL; // Desired velocity setpoint (signed)
	_Enabled		   : BOOL;
	McMoveVel1		   : MC_MoveVelocity;
	McMoveVel2		   : MC_MoveVelocity;
	McHalt			   : MC_Halt;
	Toggle			   : BOOL  := FALSE;
	LastVelocity	   : LREAL := 0.0;
	FirstCycle		   : BOOL  := TRUE;
	VelocityTolerance  : LREAL := 0.00001; // Threshold for issuing new command
	AbsVelocity		   : LREAL;
	Direction		   : MC_Direction;
	StopActive		   : BOOL := FALSE;
	_Error			   : BOOL;
	_ErrorID		   : UDINT;
	_Busy			   : BOOL;
	EnableSmoothing	   : BOOL := TRUE;	  // Enable PT1 velocity smoothing
	FilterTimeConstant : TIME := T#190MS; // PT1 time constant (tT1) - adjust for smoothing strength

	// PT1 smoothing
	PT1				: FB_CTRL_PT1;
	PT1Params		: ST_CTRL_PT1_PARAMS;
	GetCycleTime	: FB_CTRL_GET_TASK_CYCLETIME;
	PT1Initialized	: BOOL := FALSE;
	WorkingVelocity : LREAL; // The actual velocity setpoint being fed to NC (smoothed or raw)
END_VAR

{attribute 'monitoring' := 'call'}
PROPERTY Busy : BOOL
GET
Busy := _Busy;
END_GET
END_PROPERTY

METHOD CyclicLogic
// Initialize PT1 parameters once task cycle time is known
IF NOT PT1Initialized THEN
	GetCycleTime(eMode := eCTRL_MODE_ACTIVE);
	IF GetCycleTime.bCycleTimeValid THEN
		PT1Params.tTaskCycleTime := GetCycleTime.tTaskCycleTime;
		PT1Params.tCtrlCycleTime := GetCycleTime.tTaskCycleTime; // Process every cycle
		PT1Initialized			 := TRUE;
	ELSE
		// PT1 not ready yet - set defaults and exit early
		WorkingVelocity := TargetVelocity;
		RETURN;
	END_IF
END_IF

// Update PT1 parameters from inputs (allows runtime tuning)
PT1Params.fKp := 0.9;
PT1Params.tT1 := FilterTimeConstant;
// Apply velocity smoothing if enabled
IF EnableSmoothing THEN
	PT1(fIn			  := TargetVelocity,
		fManSyncValue := TargetVelocity,
		bSync		  := FALSE,
		eMode		  := eCTRL_MODE_ACTIVE,
		bHold		  := FALSE,
		stParams	  := PT1Params);

	WorkingVelocity := PT1.fOut;
ELSE
	// No smoothing - sync PT1 to current value
	PT1(fIn			  := TargetVelocity,
		fManSyncValue := TargetVelocity,
		bSync		  := TRUE, // Sync to input when smoothing disabled
		eMode		  := eCTRL_MODE_ACTIVE,
		bHold		  := FALSE,
		stParams	  := PT1Params);

	WorkingVelocity := TargetVelocity;
END_IF

// Determine if we need to issue a new velocity command
IF _Enabled THEN
	// Check if we should stop (working velocity near zero)
	IF ABS(WorkingVelocity) < VelocityTolerance THEN
		// Issue stop command if not already stopping
		IF NOT StopActive THEN
			StopActive	 := TRUE;
			LastVelocity := 0.0;
		END_IF

		// Execute stop with aborting buffer mode
		McHalt(Axis := Axis, Execute := TRUE);

		// Reset velocity FBs
		McMoveVel1(Axis := Axis, Execute := FALSE);
		McMoveVel2(Axis := Axis, Execute := FALSE);
		_Busy	 := McHalt.Busy;
		_Error	 := McHalt.Error;
		_ErrorID := McHalt.ErrorID;
	ELSE
		// We have a non-zero target velocity
		StopActive := FALSE;

		// Reset stop FB
		McHalt(Axis := Axis, Execute := FALSE);

		// Calculate absolute velocity and direction
		AbsVelocity := ABS(WorkingVelocity);
		IF WorkingVelocity >= 0.0 THEN
			Direction := MC_Positive_Direction;
		ELSE
			Direction := MC_Negative_Direction;
		END_IF

		// Check if velocity setpoint has changed significantly
		IF ABS(WorkingVelocity - LastVelocity) > VelocityTolerance OR FirstCycle THEN
			// Toggle between FB instances to achieve buffer aborting
			Toggle		 := NOT Toggle;
			LastVelocity := WorkingVelocity;
			FirstCycle	 := FALSE;
		END_IF

		// Execute alternating MoveVelocity commands with BufferMode := MC_Aborting
		McMoveVel1(Axis		  := Axis,
				   Execute	  := _Enabled AND Toggle,
				   Velocity	  := AbsVelocity,
				   Direction  := Direction,
				   BufferMode := MC_Aborting);

		McMoveVel2(Axis		  := Axis,
				   Execute	  := _Enabled AND NOT Toggle,
				   Velocity	  := AbsVelocity,
				   Direction  := Direction,
				   BufferMode := MC_Aborting);

		// Outputs
		_Busy	 := McMoveVel1.Busy OR McMoveVel2.Busy;
		_Error	 := McMoveVel1.Error OR McMoveVel2.Error;
		_ErrorID := SEL(McMoveVel1.Error, McMoveVel2.ErrorID, McMoveVel1.ErrorID);
	END_IF
ELSE
	// Reset when disabled
	McMoveVel1(Axis := Axis, Execute := FALSE);
	McMoveVel2(Axis := Axis, Execute := FALSE);
	McHalt(Axis := Axis, Execute := FALSE);
	FirstCycle := TRUE;
	StopActive := FALSE;

	// Sync PT1 to zero when disabled
	PT1(fIn			  := 0.0,
		fManSyncValue := 0.0,
		bSync		  := TRUE,
		eMode		  := eCTRL_MODE_ACTIVE,
		bHold		  := FALSE,
		stParams	  := PT1Params);

	_Busy	 := FALSE;
	_Error	 := FALSE;
	_ErrorID := 0;
END_IF
END_METHOD

METHOD Disable
_Enabled := FALSE;
END_METHOD

METHOD Enable
_Enabled := TRUE;
END_METHOD

{attribute 'monitoring' := 'call'}
PROPERTY Enabled : BOOL
GET
Enabled := _Enabled;
END_GET
END_PROPERTY

{attribute 'monitoring' := 'call'}
PROPERTY Error : BOOL
GET
Error := _Error;
END_GET
END_PROPERTY

{attribute 'monitoring' := 'call'}
PROPERTY ErrorId : UDINT
GET
ErrorId := _ErrorId;
END_GET
END_PROPERTY

(*FB_Init is always available implicitly and it is used primarily for initialization.
The return value is not evaluated. For a specific influence, you can also declare the
methods explicitly and provide additional code there with the standard initialization
code. You can evaluate the return value.*)
METHOD FB_Init : BOOL
VAR_INPUT
	(* TRUE: the retain variables are initialized (reset warm / reset cold)*)
	bInitRetains	: BOOL;
	(* TRUE: the instance will be copied to the copy code afterward (online change)   *)
	bInCopyCode	: BOOL;
	Name	: Core.T_MaxString;
    Axis		   : REFERENCE TO AXIS_REF;
END_VAR
THIS^.Axis REF= Axis;
END_METHOD

METHOD SetTargetVelocity
VAR_INPUT
	TargetVelocity : LREAL; // Desired velocity setpoint (signed)
END_VAR
THIS^.TargetVelocity := TargetVelocity;
END_METHOD

END_FUNCTION_BLOCK

// ---- Components/Encoder/Encoder_HMI.TcPOU
FUNCTION_BLOCK Encoder_HMI EXTENDS HmiFunction
VAR
	EncoderSpeed	: I_AnalogInput;
	EncoderPosition : I_AnalogInput;
END_VAR

VAR PERSISTENT
	{ attribute 'TcHmiSymbol.AddSymbol' }
	{ attribute 'TcHmiSymbol.AddSymbol.UserGroups' := '__SystemAdministrators, Admin' }
	Encoder_HMI : ST_Encoder_HMI;
END_VAR

PROPERTY Config : REFERENCE TO ST_EncoderConfig_HMI
GET
Config REF= Encoder_HMI.Config;
END_GET
END_PROPERTY

PROPERTY ControlObject : I_Base
SET
__QUERYINTERFACE(ControlObject, EncoderSpeed);
END_SET
END_PROPERTY

METHOD CyclicLogic
Encoder_HMI.Name	   := Name;
Encoder_HMI.HmiEnabled := Enabled;
IF EncoderSpeed = 0 OR EncoderPosition = 0 THEN
	RETURN;
END_IF

Encoder_HMI.ActualPosition	 := EncoderPosition.Value;
Encoder_HMI.ActualSpeed		 := EncoderSpeed.Value;
Encoder_HMI.RawValuePosition := TO_UINT(EncoderPosition.RawValue);
Encoder_HMI.RawValueSpeed	 := EncoderSpeed.RawValue;
END_METHOD

(*FB_Init is always available implicitly and it is used primarily for initialization.
The return value is not evaluated. For a specific influence, you can also declare the
methods explicitly and provide additional code there with the standard initialization
code. You can evaluate the return value.*)
METHOD FB_Init : BOOL
VAR_INPUT
	(* TRUE: the retain variables are initialized (reset warm / reset cold)*)
	bInitRetains : BOOL;

	(* TRUE: the instance will be copied to the copy code afterward (online change)   *)
	bInCopyCode		: BOOL;
	Name			: Core.T_MaxString;
	EncoderSpeed	: I_AnalogInput;
	EncoderPosition : I_AnalogInput;
END_VAR
ControlType			  := 'Encoder';
LinkObject			  := 'Encoder_HMI';
THIS^.EncoderSpeed	  := EncoderSpeed;
THIS^.EncoderPosition := EncoderPosition;
END_METHOD

END_FUNCTION_BLOCK

// ---- AMR/AmrModule_HMI.TcPOU
FUNCTION_BLOCK AmrModule_HMI EXTENDS PackMLStatemachine_HMI
VAR
	AmrModule : I_AmrModule;
	{ attribute 'TcHmiSymbol.AddSymbol' }
	{ attribute 'TcHmiSymbol.AddSymbol.UserGroups' := '__SystemAdministrators, Admin' }
	AmrModule_HMI : ST_AmrModule_HMI;
END_VAR

METHOD CyclicLogic
VAR_INST
	StartRT : R_TRIG;
	StopRT	: R_TRIG;
	ResetRT : R_TRIG;
END_VAR
IF AmrModule = 0 THEN
	RETURN;
END_IF

SUPER^.CyclicLogic();
AmrModule.Override		 := AmrModule_HMI.Override;
AmrModule.BypassScanners := AmrModule_HMI.BypassScanners;

// User buttons
Statemachine_HMI.StartPermissive := Statemachine_HMI.CurrentState = E_PMLState.Stopped;
Statemachine_HMI.StopPermissive	 := Statemachine_HMI.CurrentState <> E_PMLState.Aborted;
Statemachine_HMI.ResetPermissive := Statemachine_HMI.CurrentState = E_PMLState.Aborted;
StartRT(CLK := Statemachine_HMI.StartPressed);
IF StartRT.Q THEN
	Statemachine.ChangeState(E_PMLCommand.Start);
END_IF

StopRT(CLK := Statemachine_HMI.StopPressed);
IF StopRT.Q THEN
	IF Statemachine_HMI.CurrentState = E_PMLState.Stopped THEN
		Statemachine.ChangeState(E_PMLCommand.Abort);
	ELSE
		Statemachine.ChangeState(E_PMLCommand.Stop);
	END_IF
END_IF

ResetRT(CLK := Statemachine_HMI.ResetPressed);
IF ResetRT.Q THEN
	IF Statemachine_HMI.CurrentState = E_PMLState.Aborted THEN
		Statemachine.ChangeState(E_PMLCommand.Clear);
	ELSE
		Statemachine.ChangeState(E_PMLCommand.Reset);
	END_IF
END_IF
END_METHOD

(*FB_Init is always available implicitly and it is used primarily for initialization.
The return value is not evaluated. For a specific influence, you can also declare the
methods explicitly and provide additional code there with the standard initialization
code. You can evaluate the return value.*)
METHOD FB_Init : BOOL
VAR_INPUT
	(* TRUE: the retain variables are initialized (reset warm / reset cold)*)
	bInitRetains : BOOL;

	(* TRUE: the instance will be copied to the copy code afterward (online change)   *)
	bInCopyCode	 : BOOL;
	Name		 : Core.T_MaxString;
	Statemachine : I_Statemachine;
	AmrModule	 : I_AmrModule;
END_VAR
THIS^.AmrModule := AmrModule;
END_METHOD

END_FUNCTION_BLOCK

// ---- Components/Navitrol/HMI/Navitrol_HMI.TcPOU
FUNCTION_BLOCK Navitrol_HMI EXTENDS HmiFunction
VAR
	NavitrolStatus : I_Navitrol_Status;
	NavitrolComs   : I_TcpIpConnection;
	{ attribute 'TcHmiSymbol.AddSymbol' }
	{ attribute 'TcHmiSymbol.AddSymbol.UserGroups' := '__SystemAdministrators, Admin' }
	Navitrol_HMI : ST_Navitrol_HMI;
END_VAR

PROPERTY ControlObject : I_Base
SET
__QUERYINTERFACE(ControlObject, NavitrolComs);
END_SET
END_PROPERTY

METHOD CyclicLogic
Navitrol_HMI.HmiEnabled			 := THIS^.Enabled;
Navitrol_HMI.CommunicationActive := NavitrolComs.ConnectionState = E_SocketConnectionState.eSOCKET_CONNECTED;
Navitrol_HMI.Status				 := NavitrolStatus.NavitrolStatus.State;
END_METHOD

(*FB_Init is always available implicitly and it is used primarily for initialization.
The return value is not evaluated. For a specific influence, you can also declare the
methods explicitly and provide additional code there with the standard initialization
code. You can evaluate the return value.*)
METHOD FB_Init : BOOL
VAR_INPUT
	(* TRUE: the retain variables are initialized (reset warm / reset cold)*)
	bInitRetains : BOOL;

	(* TRUE: the instance will be copied to the copy code afterward (online change)   *)
	bInCopyCode	   : BOOL;
	Name		   : Core.T_MaxString;
	NavitrolStatus : I_Navitrol_Status;
	NavitrolComs   : I_TcpIpConnection;
END_VAR
Navitrol_HMI.Name	 := Name;
THIS^.LinkObject	 := 'Navitrol_HMI';
THIS^.ControlType	 := 'Navitrol';
THIS^.NavitrolStatus := NavitrolStatus;
THIS^.NavitrolComs	 := NavitrolComs;
END_METHOD

{attribute 'monitoring' := 'call'}
PROPERTY NavitrolHasControl : BOOL
GET
NavitrolHasControl := Navitrol_HMI.ControlFromNavitrol;
END_GET
END_PROPERTY

END_FUNCTION_BLOCK

// ---- Components/Nanotec/COEDriveControl.TcPOU
FUNCTION_BLOCK COEDriveControl
VAR_INPUT
	Enable	   : BOOL;
	Reset	   : BOOL;
	SetVelIncr : INT;
	Manual	   : BOOL;
END_VAR

VAR_OUTPUT
	Ready	   : BOOL;
	Faulted	   : BOOL;
	ActVelIncr : INT;
END_VAR

VAR
	COEStatus			  AT %I* : WORD;
	COEControl			  AT %Q* : WORD;
	ModeOfOperation		  AT %Q* : SINT := 2;
	ModeOfOperationStatus AT %I* : SINT;
	ActVel				  AT %I* : INT;
	ActPos				  AT %I* : INT;
	SetVel				  AT %Q* : INT;
	MotorTypeClosedLoop	  AT %Q* : UDINT := 65;
	SetupMode					 : BOOL;
	Seq							 : UDINT;
	WriteDelay					 : TON;
	{ attribute 'TcHmiSymbol.AddSymbol' }
	{ attribute 'TcHmiSymbol.AddSymbol.UserGroups' := '__SystemAdministrators, Admin' }
	HMI : ST_Nanotec_HMI;
END_VAR

// Interfaces with the Elmo Drive, to maintain the internal state machine (DS-402)
// Check interface document for DS-402 and Beckhoff EL7211 manual for more information
IF Manual THEN
	Enable := HMI.JogBwd OR HMI.JogFwd;
	IF HMI.JogBwd THEN
		SetVelIncr := -50;
	END_IF

	IF HMI.JogFwd THEN
		SetVelIncr := 50;
	END_IF
END_IF

HMI.Name	   := 'Lift';
HMI.ActVelIncr := ActVelIncr;
HMI.Faulted	   := Faulted;
HMI.Ready	   := Ready;
//
IF NOT SetupMode THEN
	IF (COEStatus AND 16#006F) = 16#0027 THEN (*State 4*)
		Ready := TRUE;
		IF Enable THEN
			COEControl := 16#000F;
		ELSE
			COEControl := 16#0006;
		END_IF;
	ELSIF (COEStatus AND 16#006F) = 16#0021 THEN (*State 2*)
		Ready := FALSE;
		IF Enable THEN
			COEControl := 16#0007;
		ELSIF Reset THEN
			COEControl := 16#0080;
		ELSE
			COEControl := 16#0006;
		END_IF;
	ELSIF (COEStatus AND 16#000F) = 16#0008 THEN (*State F*)
		Ready	:= FALSE;
		Faulted := TRUE;
		Enable	:= FALSE;
		IF Reset THEN
			COEControl := 16#0080;
		ELSE
			COEControl := 16#0000;
		END_IF;
	ELSIF (COEStatus AND 16#004F) = 16#0040 THEN (*State 1*) //For Elmo
		Ready	:= FALSE;
		Faulted := FALSE;
		IF Reset THEN
			COEControl := 16#0080;
		ELSE
			COEControl := 16#0006;
		END_IF;
	ELSIF (COEStatus AND 16#006F) = 16#0023 THEN (*State 3*)
		Ready := FALSE;
		IF Enable THEN
			COEControl := 16#000F;
		END_IF;
	ELSIF (COEStatus AND 16#000F) = 16#0007 THEN (*State 7*)
		Ready := FALSE;
	END_IF;

	ActVelIncr := ActVel;
	SetVel	   := SetVelIncr;
ELSE
	CASE Seq OF
		0:
			COEControl		:= 0;
			ModeOfOperation := 0;
			WriteDelay(IN := FALSE, PT := T#250MS);

		10:
			COEControl := 16#06;
			WriteDelay(IN := TRUE, PT := T#250MS);
			IF WriteDelay.Q THEN
				IF COEStatus.0 AND COEStatus.5 AND COEStatus.9 THEN
					WriteDelay(IN := FALSE);
					Seq := 20;
				END_IF
			END_IF

		20:
			ModeOfOperation := 16#FE;
			COEControl		:= 16#07;
			WriteDelay(IN := TRUE, PT := T#250MS);
			IF WriteDelay.Q THEN
				IF COEStatus.0 AND COEStatus.1 AND COEStatus.4 AND COEStatus.5 AND COEStatus.9 THEN
					WriteDelay(IN := FALSE);
					Seq := 30;
				END_IF
			END_IF

		30:
			COEControl := 16#0F;
			WriteDelay(IN := TRUE, PT := T#250MS);
			IF WriteDelay.Q THEN
				IF COEStatus.0 AND COEStatus.1 AND COEStatus.2 AND COEStatus.4 AND COEStatus.5 AND COEStatus.9 THEN
					WriteDelay(IN := FALSE);
					Seq := 40;
				END_IF
			END_IF

		40:
			IF ModeOfOperationStatus = -2 THEN
				Seq := 50;
			END_IF

		50:
			COEControl := 16#1F;
			IF COEStatus.0 AND COEStatus.1 AND COEStatus.2 AND COEStatus.4 AND COEStatus.5 AND COEStatus.9 AND COEStatus.12 THEN
				WriteDelay(IN := FALSE);
				Seq := 60;
			END_IF
	END_CASE
END_IF

END_FUNCTION_BLOCK

// ---- Components/DEGREE_TO_RADIAN.TcPOU
FUNCTION DEGREE_TO_RADIAN : LREAL
VAR_INPUT
	Degree : LREAL;
END_VAR

DEGREE_TO_RADIAN := Degree * (PI / 180.0);

END_FUNCTION
